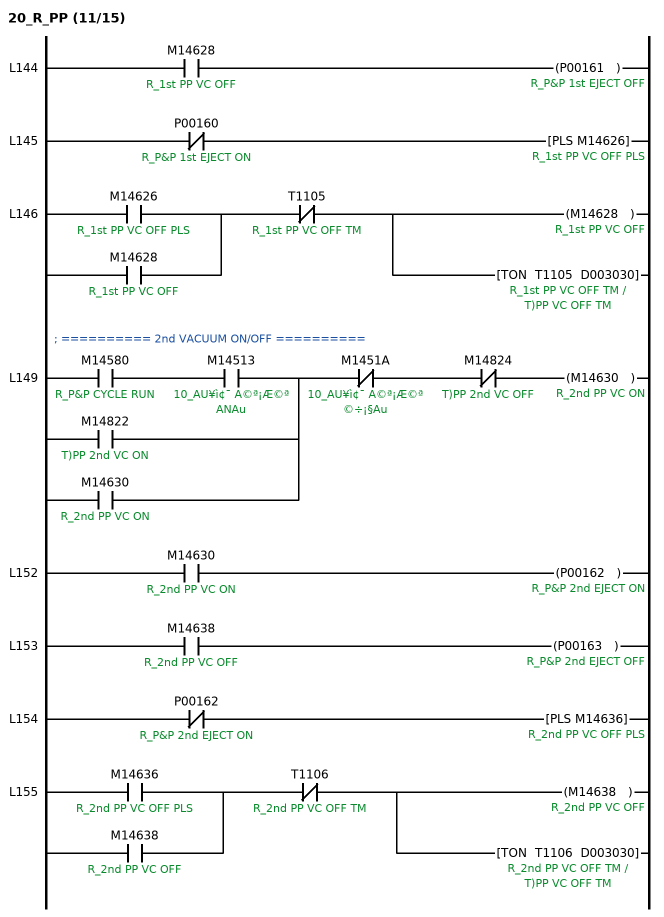
[picture p192: 20_R_PP rungs L144-L155]
; L144
LOAD      M14628	// R_1st PP VC OFF
OUT       P00161	// R_P&P 1st EJECT OFF
; L145
LOAD NOT  P00160	// R_P&P 1st EJECT ON
OUTP      M14626	// R_1st PP VC OFF PLS
; L146
LOAD      M14626	// R_1st PP VC OFF PLS
OR        M14628	// R_1st PP VC OFF
AND NOT   T1105	// R_1st PP VC OFF TM
OUT       M14628	// R_1st PP VC OFF
TON       T1105 D003030	// R_1st PP VC OFF TM / T)PP VC OFF TM
// ========== 2nd VACUUM ON/OFF ==========
; L149
LOAD      M14580	// R_P&P CYCLE RUN
AND       M14513	// 10_AU¥ì¢¯ A©ª¡Æ©ª ANAu
OR        M14822	// T)PP 2nd VC ON
OR        M14630	// R_2nd PP VC ON
AND NOT   M1451A	// 10_AU¥ì¢¯ A©ª¡Æ©ª ©÷¡§Au
AND NOT   M14824	// T)PP 2nd VC OFF
OUT       M14630	// R_2nd PP VC ON
; L152
LOAD      M14630	// R_2nd PP VC ON
OUT       P00162	// R_P&P 2nd EJECT ON
; L153
LOAD      M14638	// R_2nd PP VC OFF
OUT       P00163	// R_P&P 2nd EJECT OFF
; L154
LOAD NOT  P00162	// R_P&P 2nd EJECT ON
OUTP      M14636	// R_2nd PP VC OFF PLS
; L155
LOAD      M14636	// R_2nd PP VC OFF PLS
OR        M14638	// R_2nd PP VC OFF
AND NOT   T1106	// R_2nd PP VC OFF TM
OUT       M14638	// R_2nd PP VC OFF
TON       T1106 D003030	// R_2nd PP VC OFF TM / T)PP VC OFF TM

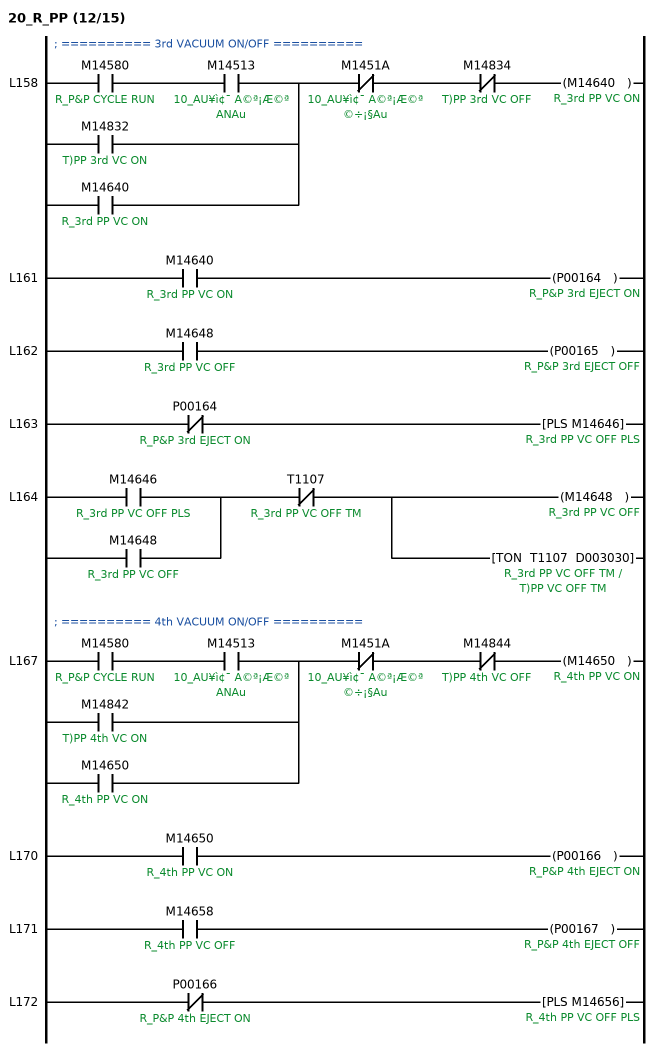
// ========== 3rd VACUUM ON/OFF ==========
; L158
LOAD      M14580	// R_P&P CYCLE RUN
AND       M14513	// 10_AU¥ì¢¯ A©ª¡Æ©ª ANAu
OR        M14832	// T)PP 3rd VC ON
OR        M14640	// R_3rd PP VC ON
AND NOT   M1451A	// 10_AU¥ì¢¯ A©ª¡Æ©ª ©÷¡§Au
AND NOT   M14834	// T)PP 3rd VC OFF
OUT       M14640	// R_3rd PP VC ON
; L161
LOAD      M14640	// R_3rd PP VC ON
OUT       P00164	// R_P&P 3rd EJECT ON
; L162
LOAD      M14648	// R_3rd PP VC OFF
OUT       P00165	// R_P&P 3rd EJECT OFF
; L163
LOAD NOT  P00164	// R_P&P 3rd EJECT ON
OUTP      M14646	// R_3rd PP VC OFF PLS
; L164
LOAD      M14646	// R_3rd PP VC OFF PLS
OR        M14648	// R_3rd PP VC OFF
AND NOT   T1107	// R_3rd PP VC OFF TM
OUT       M14648	// R_3rd PP VC OFF
TON       T1107 D003030	// R_3rd PP VC OFF TM / T)PP VC OFF TM
// ========== 4th VACUUM ON/OFF ==========
; L167
LOAD      M14580	// R_P&P CYCLE RUN
AND       M14513	// 10_AU¥ì¢¯ A©ª¡Æ©ª ANAu
OR        M14842	// T)PP 4th VC ON
OR        M14650	// R_4th PP VC ON
AND NOT   M1451A	// 10_AU¥ì¢¯ A©ª¡Æ©ª ©÷¡§Au
AND NOT   M14844	// T)PP 4th VC OFF
OUT       M14650	// R_4th PP VC ON
; L170
LOAD      M14650	// R_4th PP VC ON
OUT       P00166	// R_P&P 4th EJECT ON
; L171
LOAD      M14658	// R_4th PP VC OFF
OUT       P00167	// R_P&P 4th EJECT OFF
; L172
LOAD NOT  P00166	// R_P&P 4th EJECT ON
OUTP      M14656	// R_4th PP VC OFF PLS

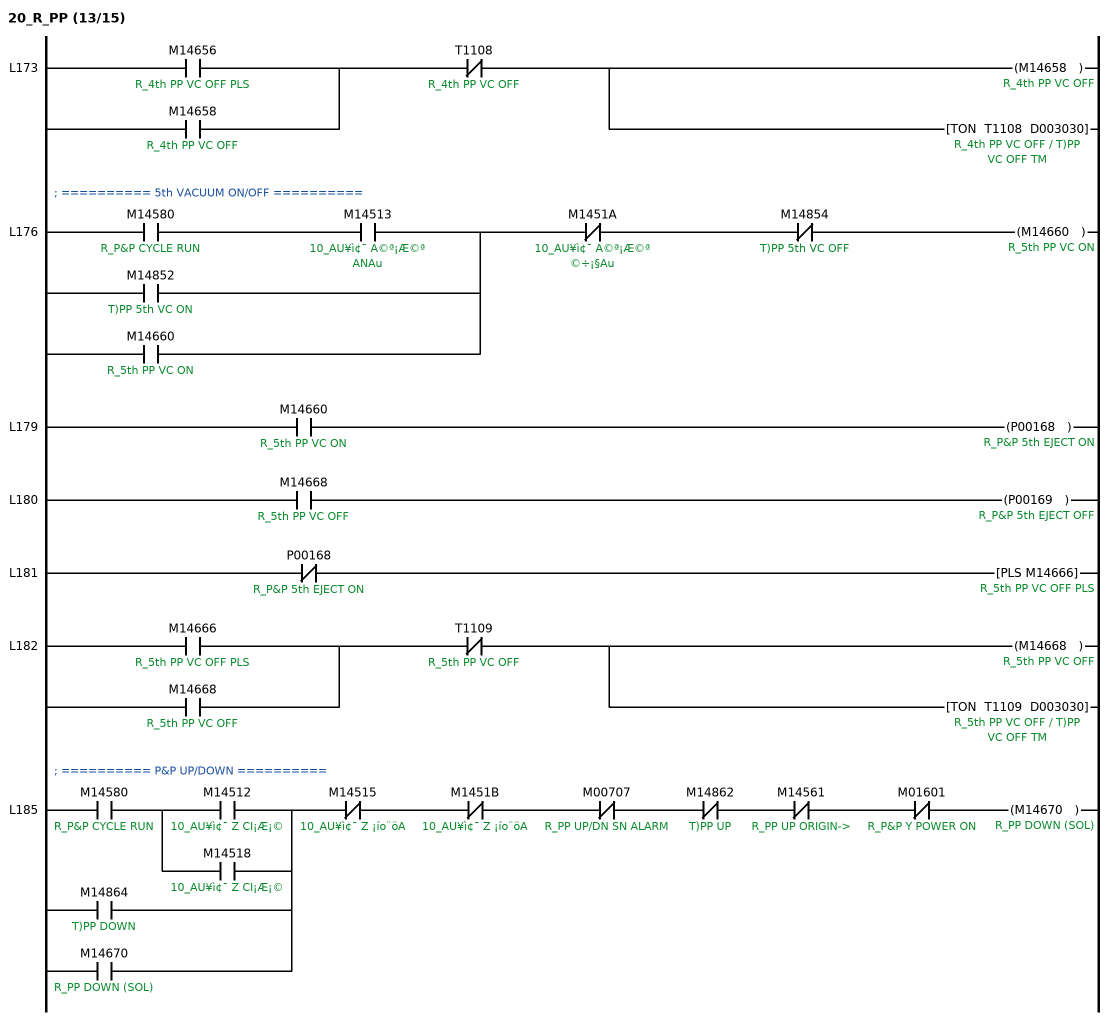
; L173
LOAD      M14656	// R_4th PP VC OFF PLS
OR        M14658	// R_4th PP VC OFF
AND NOT   T1108	// R_4th PP VC OFF
OUT       M14658	// R_4th PP VC OFF
TON       T1108 D003030	// R_4th PP VC OFF / T)PP VC OFF TM
// ========== 5th VACUUM ON/OFF ==========
; L176
LOAD      M14580	// R_P&P CYCLE RUN
AND       M14513	// 10_AU¥ì¢¯ A©ª¡Æ©ª ANAu
OR        M14852	// T)PP 5th VC ON
OR        M14660	// R_5th PP VC ON
AND NOT   M1451A	// 10_AU¥ì¢¯ A©ª¡Æ©ª ©÷¡§Au
AND NOT   M14854	// T)PP 5th VC OFF
OUT       M14660	// R_5th PP VC ON
; L179
LOAD      M14660	// R_5th PP VC ON
OUT       P00168	// R_P&P 5th EJECT ON
; L180
LOAD      M14668	// R_5th PP VC OFF
OUT       P00169	// R_P&P 5th EJECT OFF
; L181
LOAD NOT  P00168	// R_P&P 5th EJECT ON
OUTP      M14666	// R_5th PP VC OFF PLS
; L182
LOAD      M14666	// R_5th PP VC OFF PLS
OR        M14668	// R_5th PP VC OFF
AND NOT   T1109	// R_5th PP VC OFF
OUT       M14668	// R_5th PP VC OFF
TON       T1109 D003030	// R_5th PP VC OFF / T)PP VC OFF TM
// ========== P&P UP/DOWN ==========
; L185
LOAD      M14580	// R_P&P CYCLE RUN
LOAD      M14512	// 10_AU¥ì¢¯ Z CI¡Æ¡©
OR        M14518	// 10_AU¥ì¢¯ Z CI¡Æ¡©
AND LOAD
OR        M14864	// T)PP DOWN
OR        M14670	// R_PP DOWN (SOL)
AND NOT   M14515	// 10_AU¥ì¢¯ Z ¡ío¨öA
AND NOT   M1451B	// 10_AU¥ì¢¯ Z ¡ío¨öA
AND NOT   M00707	// R_PP UP/DN SN ALARM
AND NOT   M14862	// T)PP UP
AND NOT   M14561	// R_PP UP ORIGIN->
AND NOT   M01601	// R_P&P Y POWER ON
OUT       M14670	// R_PP DOWN (SOL)

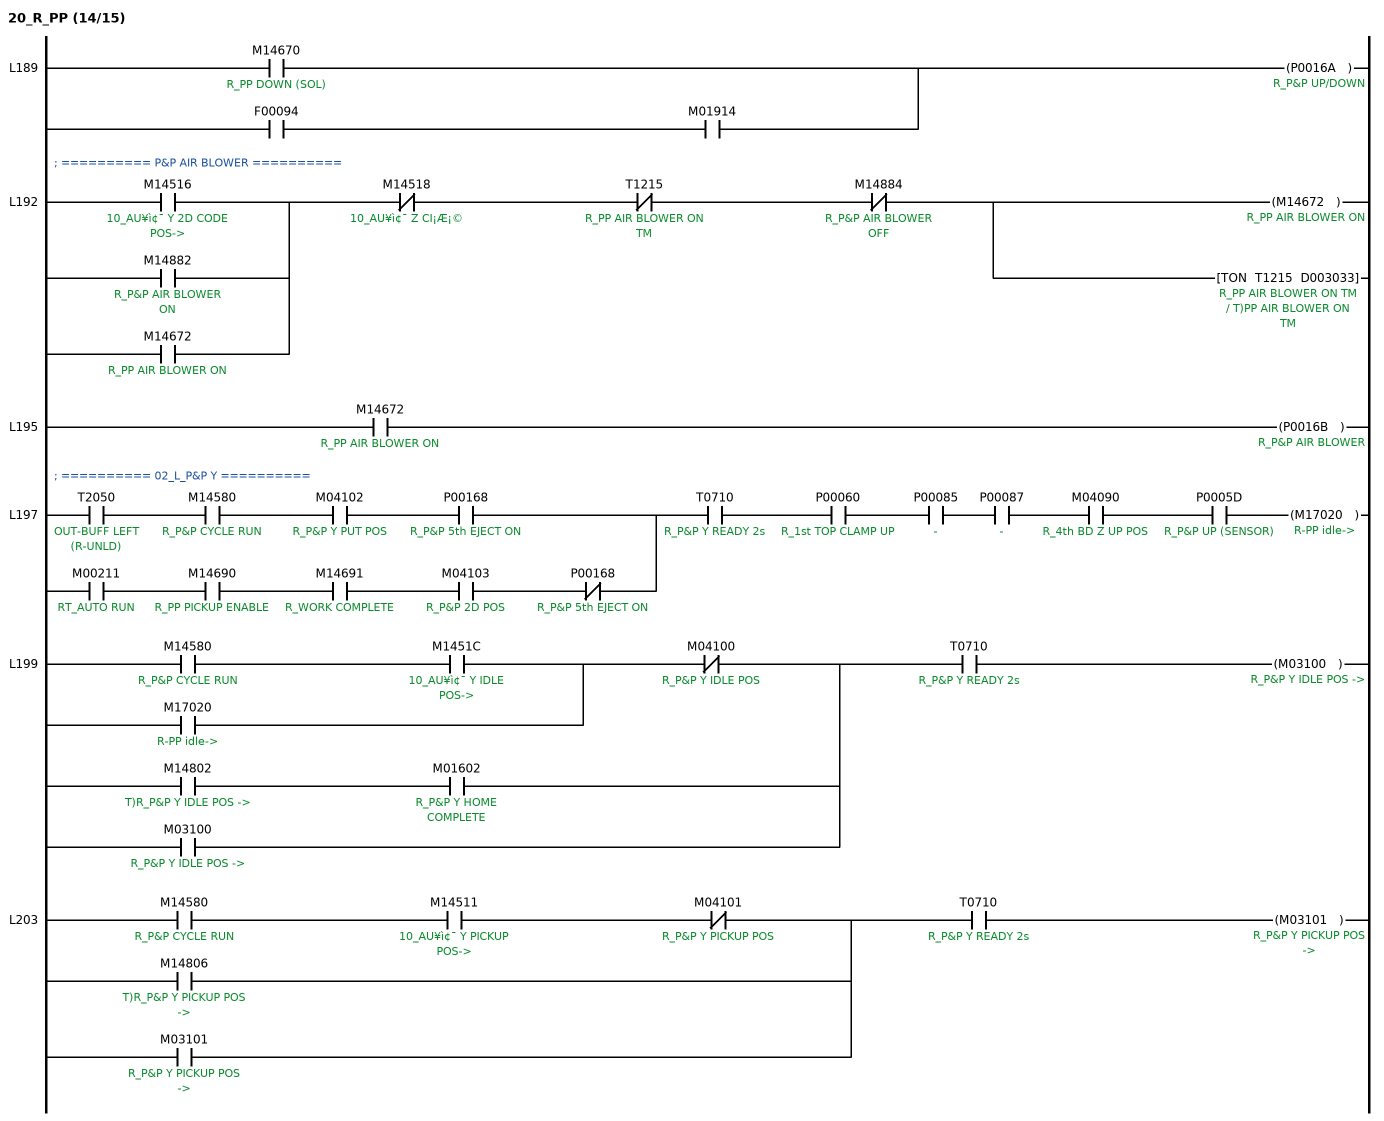
; L189
LOAD      M14670	// R_PP DOWN (SOL)
LOAD      F00094
AND       M01914
OR LOAD
OUT       P0016A	// R_P&P UP/DOWN
// ========== P&P AIR BLOWER ==========
; L192
LOAD      M14516	// 10_AU¥ì¢¯ Y 2D CODE POS->
OR        M14882	// R_P&P AIR BLOWER ON
OR        M14672	// R_PP AIR BLOWER ON
AND NOT   M14518	// 10_AU¥ì¢¯ Z CI¡Æ¡©
AND NOT   T1215	// R_PP AIR BLOWER ON TM
AND NOT   M14884	// R_P&P AIR BLOWER OFF
OUT       M14672	// R_PP AIR BLOWER ON
TON       T1215 D003033	// R_PP AIR BLOWER ON TM / T)PP AIR BLOWER ON TM
; L195
LOAD      M14672	// R_PP AIR BLOWER ON
OUT       P0016B	// R_P&P AIR BLOWER
// ========== 02_L_P&P Y ==========
; L197
LOAD      T2050	// OUT-BUFF LEFT (R-UNLD)
AND       M14580	// R_P&P CYCLE RUN
AND       M04102	// R_P&P Y PUT POS
AND       P00168	// R_P&P 5th EJECT ON
LOAD      M00211	// RT_AUTO RUN
AND       M14690	// R_PP PICKUP ENABLE
AND       M14691	// R_WORK COMPLETE
AND       M04103	// R_P&P 2D POS
AND NOT   P00168	// R_P&P 5th EJECT ON
OR LOAD
AND       T0710	// R_P&P Y READY 2s
AND       P00060	// R_1st TOP CLAMP UP
AND       P00085	// -
AND       P00087	// -
AND       M04090	// R_4th BD Z UP POS
AND       P0005D	// R_P&P UP (SENSOR)
OUT       M17020	// R-PP idle->
; L199
LOAD      M14580	// R_P&P CYCLE RUN
AND       M1451C	// 10_AU¥ì¢¯ Y IDLE POS->
OR        M17020	// R-PP idle->
AND NOT   M04100	// R_P&P Y IDLE POS
LOAD      M14802	// T)R_P&P Y IDLE POS ->
AND       M01602	// R_P&P Y HOME COMPLETE
OR LOAD
OR        M03100	// R_P&P Y IDLE POS ->
AND       T0710	// R_P&P Y READY 2s
OUT       M03100	// R_P&P Y IDLE POS ->
; L203
LOAD      M14580	// R_P&P CYCLE RUN
AND       M14511	// 10_AU¥ì¢¯ Y PICKUP POS->
AND NOT   M04101	// R_P&P Y PICKUP POS
OR        M14806	// T)R_P&P Y PICKUP POS ->
OR        M03101	// R_P&P Y PICKUP POS ->
AND       T0710	// R_P&P Y READY 2s
OUT       M03101	// R_P&P Y PICKUP POS ->

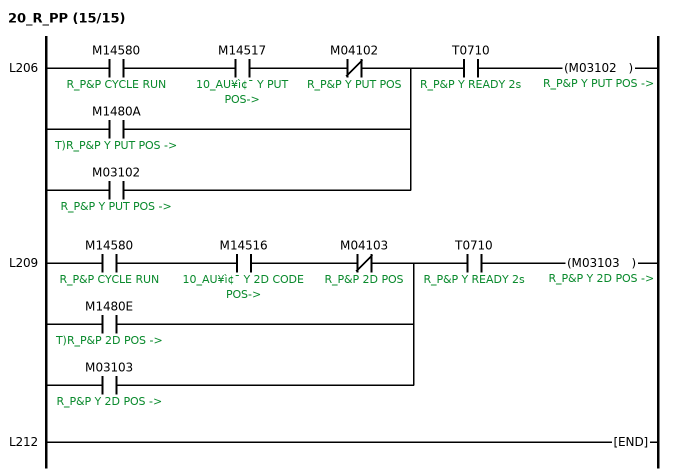
; L206
LOAD      M14580	// R_P&P CYCLE RUN
AND       M14517	// 10_AU¥ì¢¯ Y PUT POS->
AND NOT   M04102	// R_P&P Y PUT POS
OR        M1480A	// T)R_P&P Y PUT POS ->
OR        M03102	// R_P&P Y PUT POS ->
AND       T0710	// R_P&P Y READY 2s
OUT       M03102	// R_P&P Y PUT POS ->
; L209
LOAD      M14580	// R_P&P CYCLE RUN
AND       M14516	// 10_AU¥ì¢¯ Y 2D CODE POS->
AND NOT   M04103	// R_P&P 2D POS
OR        M1480E	// T)R_P&P 2D POS ->
OR        M03103	// R_P&P Y 2D POS ->
AND       T0710	// R_P&P Y READY 2s
OUT       M03103	// R_P&P Y 2D POS ->
; L212
END

PROGRAM 30_IN_LR_BUFFER (task: ¨ö¨¬A¥ì CA¡¤I¡¾¡¿¡¤¡Í)

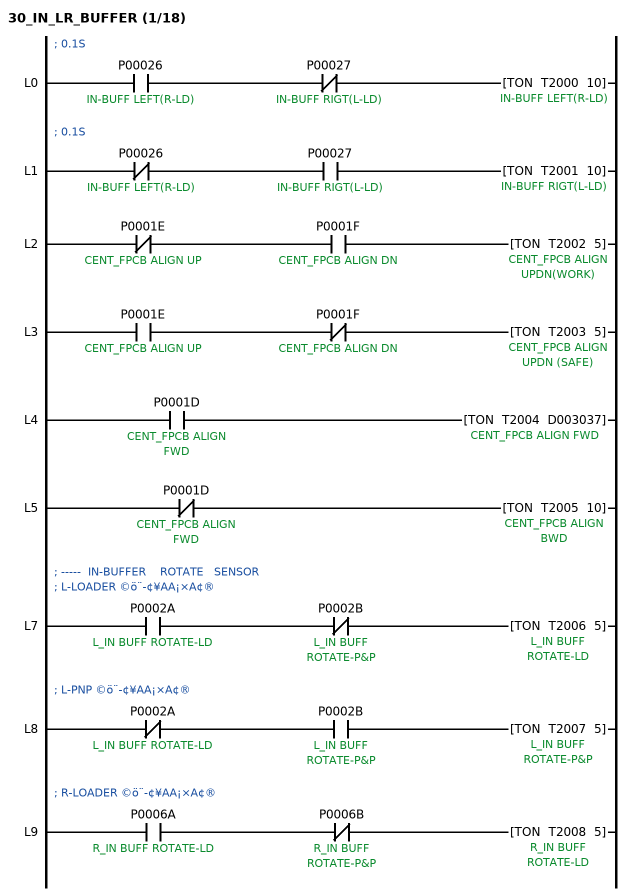
; L0
LOAD      P00026	// IN-BUFF LEFT(R-LD)
AND NOT   P00027	// IN-BUFF RIGT(L-LD)
TON       T2000 10	// IN-BUFF LEFT(R-LD)
// output comment: 0.1S
; L1
LOAD NOT  P00026	// IN-BUFF LEFT(R-LD)
AND       P00027	// IN-BUFF RIGT(L-LD)
TON       T2001 10	// IN-BUFF RIGT(L-LD)
// output comment: 0.1S
; L2
LOAD NOT  P0001E	// CENT_FPCB ALIGN UP
AND       P0001F	// CENT_FPCB ALIGN DN
TON       T2002 5	// CENT_FPCB ALIGN UPDN(WORK)
; L3
LOAD      P0001E	// CENT_FPCB ALIGN UP
AND NOT   P0001F	// CENT_FPCB ALIGN DN
TON       T2003 5	// CENT_FPCB ALIGN UPDN (SAFE)
; L4
LOAD      P0001D	// CENT_FPCB ALIGN FWD
TON       T2004 D003037	// CENT_FPCB ALIGN FWD
; L5
LOAD NOT  P0001D	// CENT_FPCB ALIGN FWD
TON       T2005 10	// CENT_FPCB ALIGN BWD
// -----  IN-BUFFER    ROTATE   SENSOR
; L7
LOAD      P0002A	// L_IN BUFF ROTATE-LD
AND NOT   P0002B	// L_IN BUFF ROTATE-P&P
TON       T2006 5	// L_IN BUFF ROTATE-LD
// output comment: L-LOADER ©ö¨­¢¥AA¡×A¢®
; L8
LOAD NOT  P0002A	// L_IN BUFF ROTATE-LD
AND       P0002B	// L_IN BUFF ROTATE-P&P
TON       T2007 5	// L_IN BUFF ROTATE-P&P
// output comment: L-PNP ©ö¨­¢¥AA¡×A¢®
; L9
LOAD      P0006A	// R_IN BUFF ROTATE-LD
AND NOT   P0006B	// R_IN BUFF ROTATE-P&P
TON       T2008 5	// R_IN BUFF ROTATE-LD
// output comment: R-LOADER ©ö¨­¢¥AA¡×A¢®

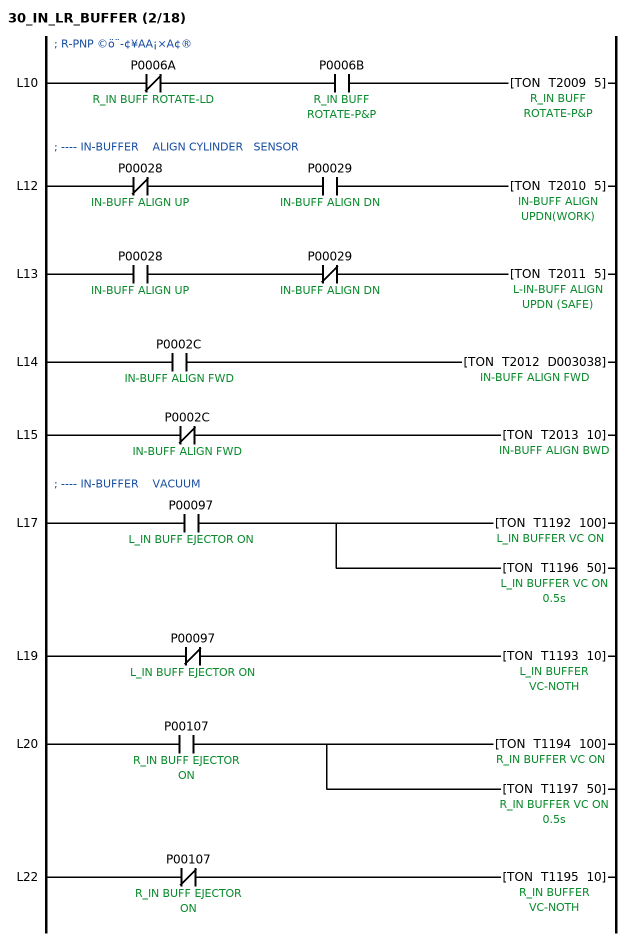
; L10
LOAD NOT  P0006A	// R_IN BUFF ROTATE-LD
AND       P0006B	// R_IN BUFF ROTATE-P&P
TON       T2009 5	// R_IN BUFF ROTATE-P&P
// output comment: R-PNP ©ö¨­¢¥AA¡×A¢®
// ---- IN-BUFFER    ALIGN CYLINDER   SENSOR
; L12
LOAD NOT  P00028	// IN-BUFF ALIGN UP
AND       P00029	// IN-BUFF ALIGN DN
TON       T2010 5	// IN-BUFF ALIGN UPDN(WORK)
; L13
LOAD      P00028	// IN-BUFF ALIGN UP
AND NOT   P00029	// IN-BUFF ALIGN DN
TON       T2011 5	// L-IN-BUFF ALIGN UPDN (SAFE)
; L14
LOAD      P0002C	// IN-BUFF ALIGN FWD
TON       T2012 D003038	// IN-BUFF ALIGN FWD
; L15
LOAD NOT  P0002C	// IN-BUFF ALIGN FWD
TON       T2013 10	// IN-BUFF ALIGN BWD
// ---- IN-BUFFER    VACUUM
; L17
LOAD      P00097	// L_IN BUFF EJECTOR ON
TON       T1192 100	// L_IN BUFFER VC ON
TON       T1196 50	// L_IN BUFFER VC ON 0.5s
; L19
LOAD NOT  P00097	// L_IN BUFF EJECTOR ON
TON       T1193 10	// L_IN BUFFER VC-NOTH
; L20
LOAD      P00107	// R_IN BUFF EJECTOR ON
TON       T1194 100	// R_IN BUFFER VC ON
TON       T1197 50	// R_IN BUFFER VC ON 0.5s
; L22
LOAD NOT  P00107	// R_IN BUFF EJECTOR ON
TON       T1195 10	// R_IN BUFFER VC-NOTH

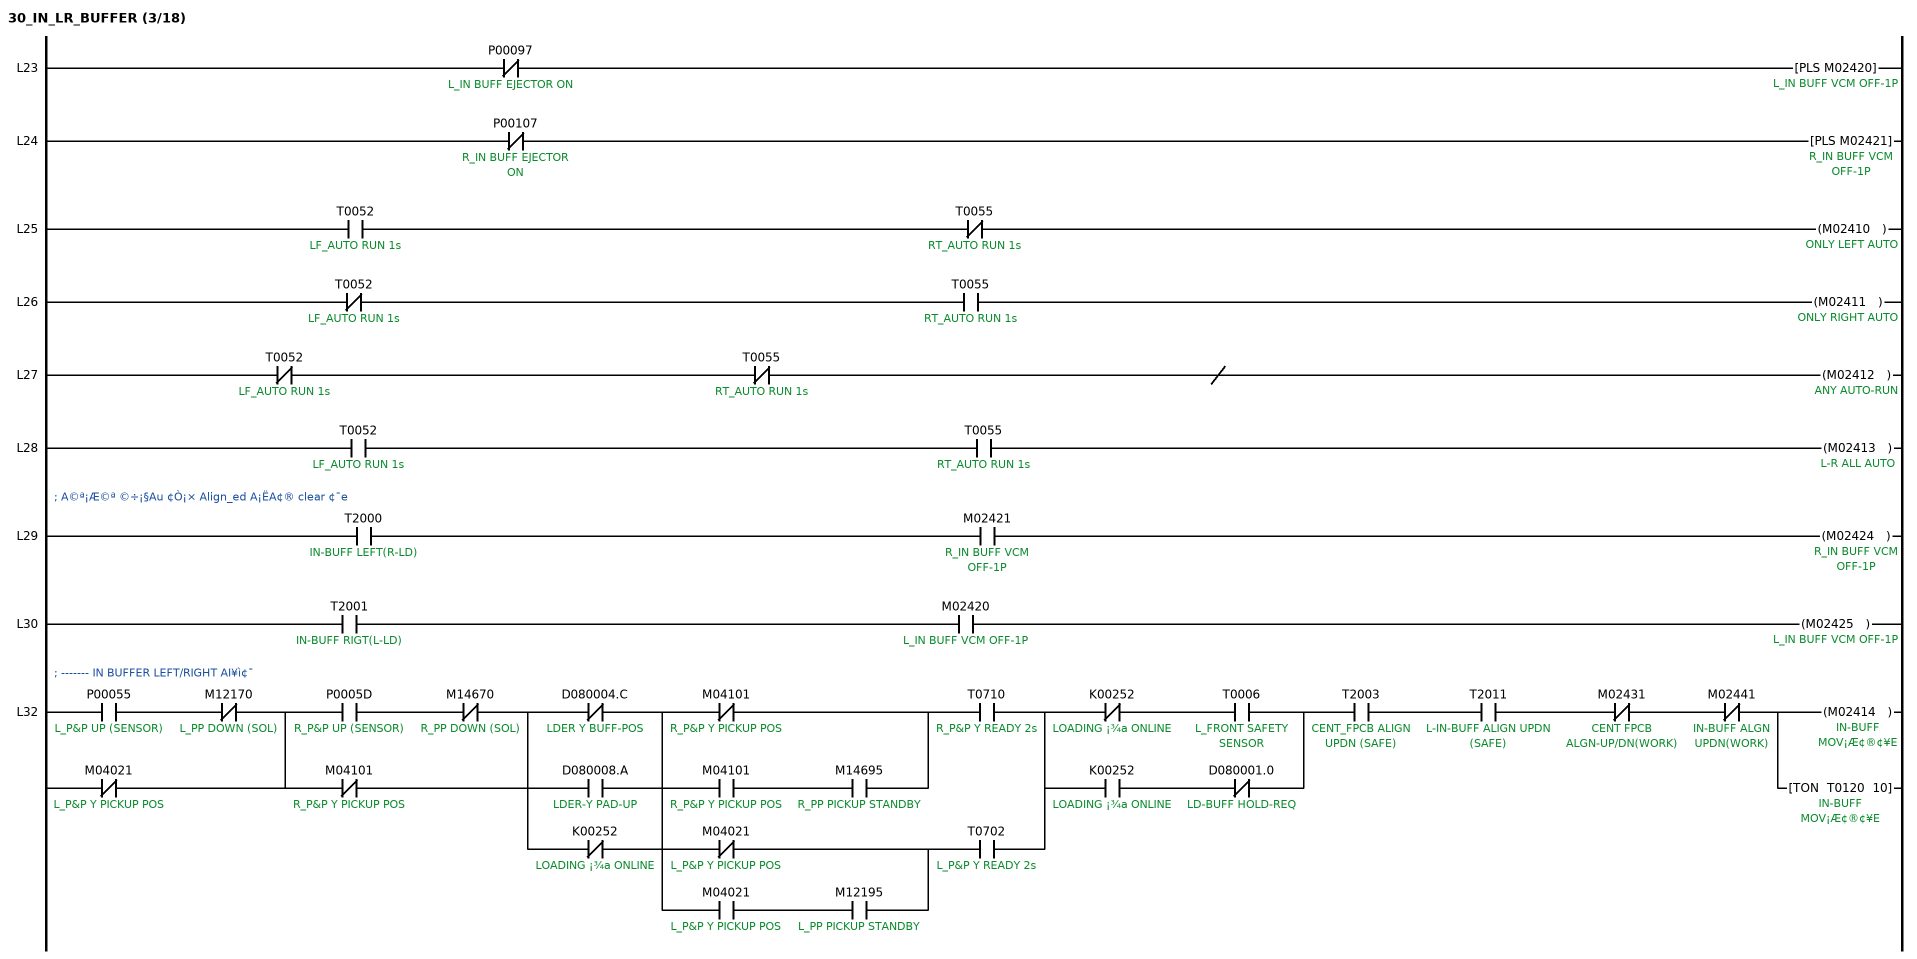
; L23
LOAD NOT  P00097	// L_IN BUFF EJECTOR ON
OUTP      M02420	// L_IN BUFF VCM OFF-1P
; L24
LOAD NOT  P00107	// R_IN BUFF EJECTOR ON
OUTP      M02421	// R_IN BUFF VCM OFF-1P
; L25
LOAD      T0052	// LF_AUTO RUN 1s
AND NOT   T0055	// RT_AUTO RUN 1s
OUT       M02410	// ONLY LEFT AUTO
; L26
LOAD NOT  T0052	// LF_AUTO RUN 1s
AND       T0055	// RT_AUTO RUN 1s
OUT       M02411	// ONLY RIGHT AUTO
; L27
LOAD NOT  T0052	// LF_AUTO RUN 1s
AND NOT   T0055	// RT_AUTO RUN 1s
NOT
OUT       M02412	// ANY AUTO-RUN
; L28
LOAD      T0052	// LF_AUTO RUN 1s
AND       T0055	// RT_AUTO RUN 1s
OUT       M02413	// L-R ALL AUTO
; L29
LOAD      T2000	// IN-BUFF LEFT(R-LD)
AND       M02421	// R_IN BUFF VCM OFF-1P
OUT       M02424	// R_IN BUFF VCM OFF-1P
// output comment: A©ª¡Æ©ª ©÷¡§Au ¢Ò¡× Align_ed A¡ËA¢® clear ¢¯e
; L30
LOAD      T2001	// IN-BUFF RIGT(L-LD)
AND       M02420	// L_IN BUFF VCM OFF-1P
OUT       M02425	// L_IN BUFF VCM OFF-1P
// ------- IN BUFFER LEFT/RIGHT AI¥ì¢¯
; L32
LOAD      P00055	// L_P&P UP (SENSOR)
AND NOT   M12170	// L_PP DOWN (SOL)
OR NOT    M04021	// L_P&P Y PICKUP POS
LOAD      P0005D	// R_P&P UP (SENSOR)
AND NOT   M14670	// R_PP DOWN (SOL)
OR NOT    M04101	// R_P&P Y PICKUP POS
AND LOAD
LOAD NOT  D080004.C	// LDER Y BUFF-POS
OR        D080008.A	// LDER-Y PAD-UP
OR NOT    K00252	// LOADING ¡¾a ONLINE
AND LOAD
LOAD NOT  M04101	// R_P&P Y PICKUP POS
LOAD      M04101	// R_P&P Y PICKUP POS
AND       M14695	// R_PP PICKUP STANDBY
OR LOAD
AND       T0710	// R_P&P Y READY 2s
LOAD NOT  M04021	// L_P&P Y PICKUP POS
LOAD      M04021	// L_P&P Y PICKUP POS
AND       M12195	// L_PP PICKUP STANDBY
OR LOAD
AND       T0702	// L_P&P Y READY 2s
OR LOAD
AND LOAD
LOAD NOT  K00252	// LOADING ¡¾a ONLINE
AND       T0006	// L_FRONT SAFETY SENSOR
LOAD      K00252	// LOADING ¡¾a ONLINE
AND NOT   D080001.0	// LD-BUFF HOLD-REQ
OR LOAD
AND LOAD
AND       T2003	// CENT_FPCB ALIGN UPDN (SAFE)
AND       T2011	// L-IN-BUFF ALIGN UPDN (SAFE)
AND NOT   M02431	// CENT FPCB ALGN-UP/DN(WORK)
AND NOT   M02441	// IN-BUFF ALGN UPDN(WORK)
OUT       M02414	// IN-BUFF MOV¡Æ¢®¢¥E
TON       T0120 10	// IN-BUFF MOV¡Æ¢®¢¥E

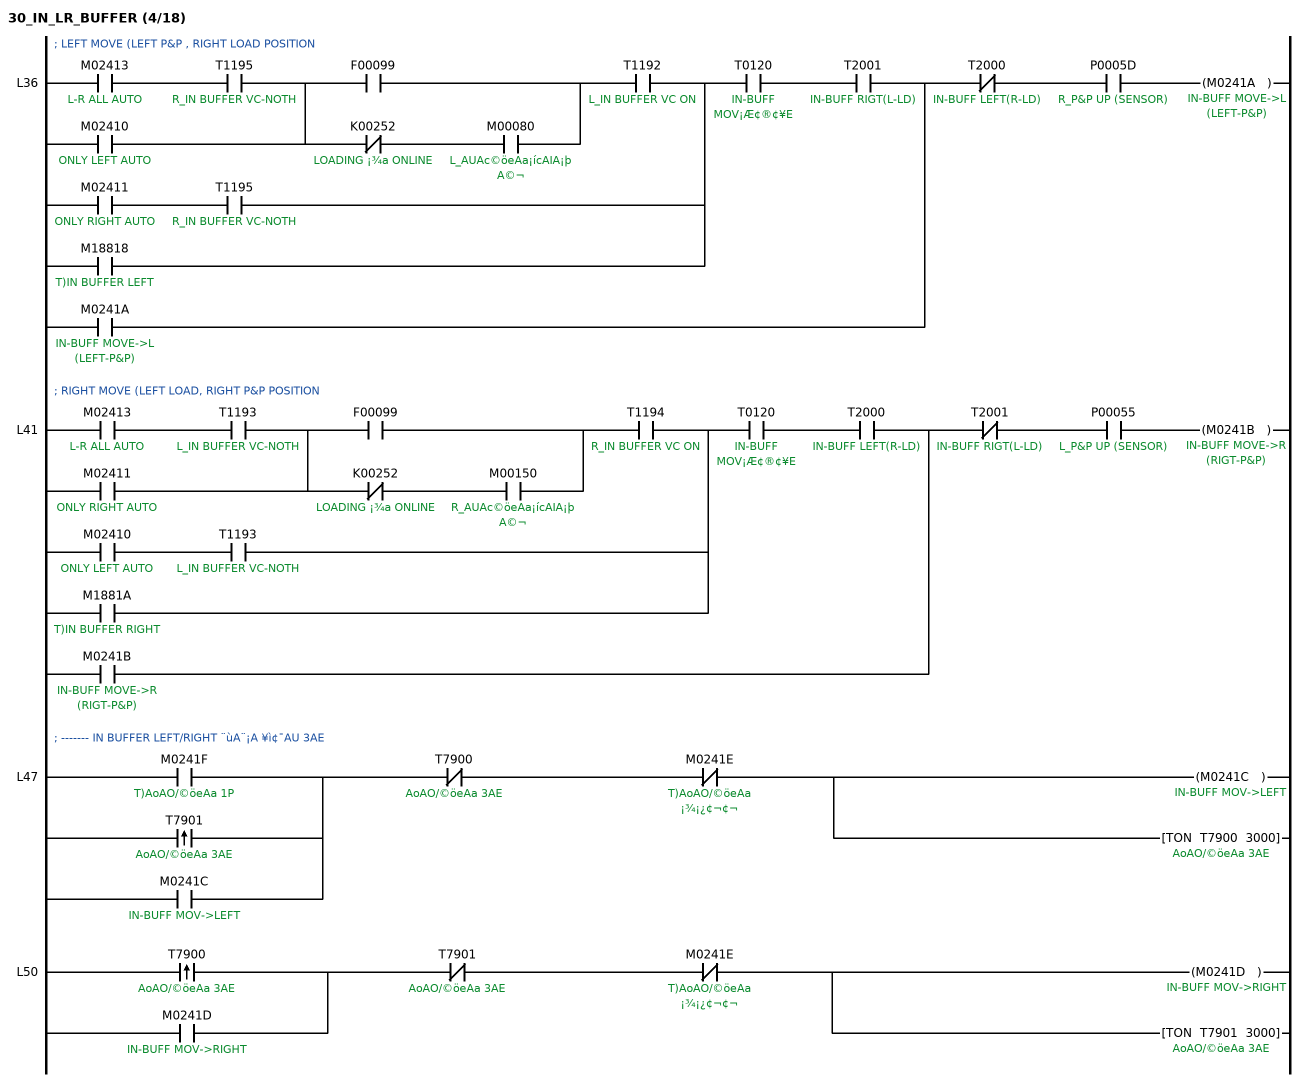
; L36
LOAD      M02413	// L-R ALL AUTO
AND       T1195	// R_IN BUFFER VC-NOTH
OR        M02410	// ONLY LEFT AUTO
LOAD      F00099
LOAD NOT  K00252	// LOADING ¡¾a ONLINE
AND       M00080	// L_AUAc©öeAa¡ícAIA¡þA©¬
OR LOAD
AND LOAD
AND       T1192	// L_IN BUFFER VC ON
LOAD      M02411	// ONLY RIGHT AUTO
AND       T1195	// R_IN BUFFER VC-NOTH
OR LOAD
OR        M18818	// T)IN BUFFER LEFT
AND       T0120	// IN-BUFF MOV¡Æ¢®¢¥E
AND       T2001	// IN-BUFF RIGT(L-LD)
OR        M0241A	// IN-BUFF MOVE->L (LEFT-P&P)
AND NOT   T2000	// IN-BUFF LEFT(R-LD)
AND       P0005D	// R_P&P UP (SENSOR)
OUT       M0241A	// IN-BUFF MOVE->L (LEFT-P&P)
// output comment: LEFT MOVE (LEFT P&P , RIGHT LOAD POSITION
; L41
LOAD      M02413	// L-R ALL AUTO
AND       T1193	// L_IN BUFFER VC-NOTH
OR        M02411	// ONLY RIGHT AUTO
LOAD      F00099
LOAD NOT  K00252	// LOADING ¡¾a ONLINE
AND       M00150	// R_AUAc©öeAa¡ícAIA¡þA©¬
OR LOAD
AND LOAD
AND       T1194	// R_IN BUFFER VC ON
LOAD      M02410	// ONLY LEFT AUTO
AND       T1193	// L_IN BUFFER VC-NOTH
OR LOAD
OR        M1881A	// T)IN BUFFER RIGHT
AND       T0120	// IN-BUFF MOV¡Æ¢®¢¥E
AND       T2000	// IN-BUFF LEFT(R-LD)
OR        M0241B	// IN-BUFF MOVE->R (RIGT-P&P)
AND NOT   T2001	// IN-BUFF RIGT(L-LD)
AND       P00055	// L_P&P UP (SENSOR)
OUT       M0241B	// IN-BUFF MOVE->R (RIGT-P&P)
// output comment: RIGHT MOVE (LEFT LOAD, RIGHT P&P POSITION
// ------- IN BUFFER LEFT/RIGHT ¨ùA¨¡A ¥ì¢¯AU 3AE
; L47
LOAD      M0241F	// T)AoAO/©öeAa 1P
ORP       T7901	// AoAO/©öeAa 3AE
OR        M0241C	// IN-BUFF MOV->LEFT
AND NOT   T7900	// AoAO/©öeAa 3AE
AND NOT   M0241E	// T)AoAO/©öeAa ¡¾¡¿¢¬¢¬
OUT       M0241C	// IN-BUFF MOV->LEFT
TON       T7900 3000	// AoAO/©öeAa 3AE
; L50
LOADP     T7900	// AoAO/©öeAa 3AE
OR        M0241D	// IN-BUFF MOV->RIGHT
AND NOT   T7901	// AoAO/©öeAa 3AE
AND NOT   M0241E	// T)AoAO/©öeAa ¡¾¡¿¢¬¢¬
OUT       M0241D	// IN-BUFF MOV->RIGHT
TON       T7901 3000	// AoAO/©öeAa 3AE

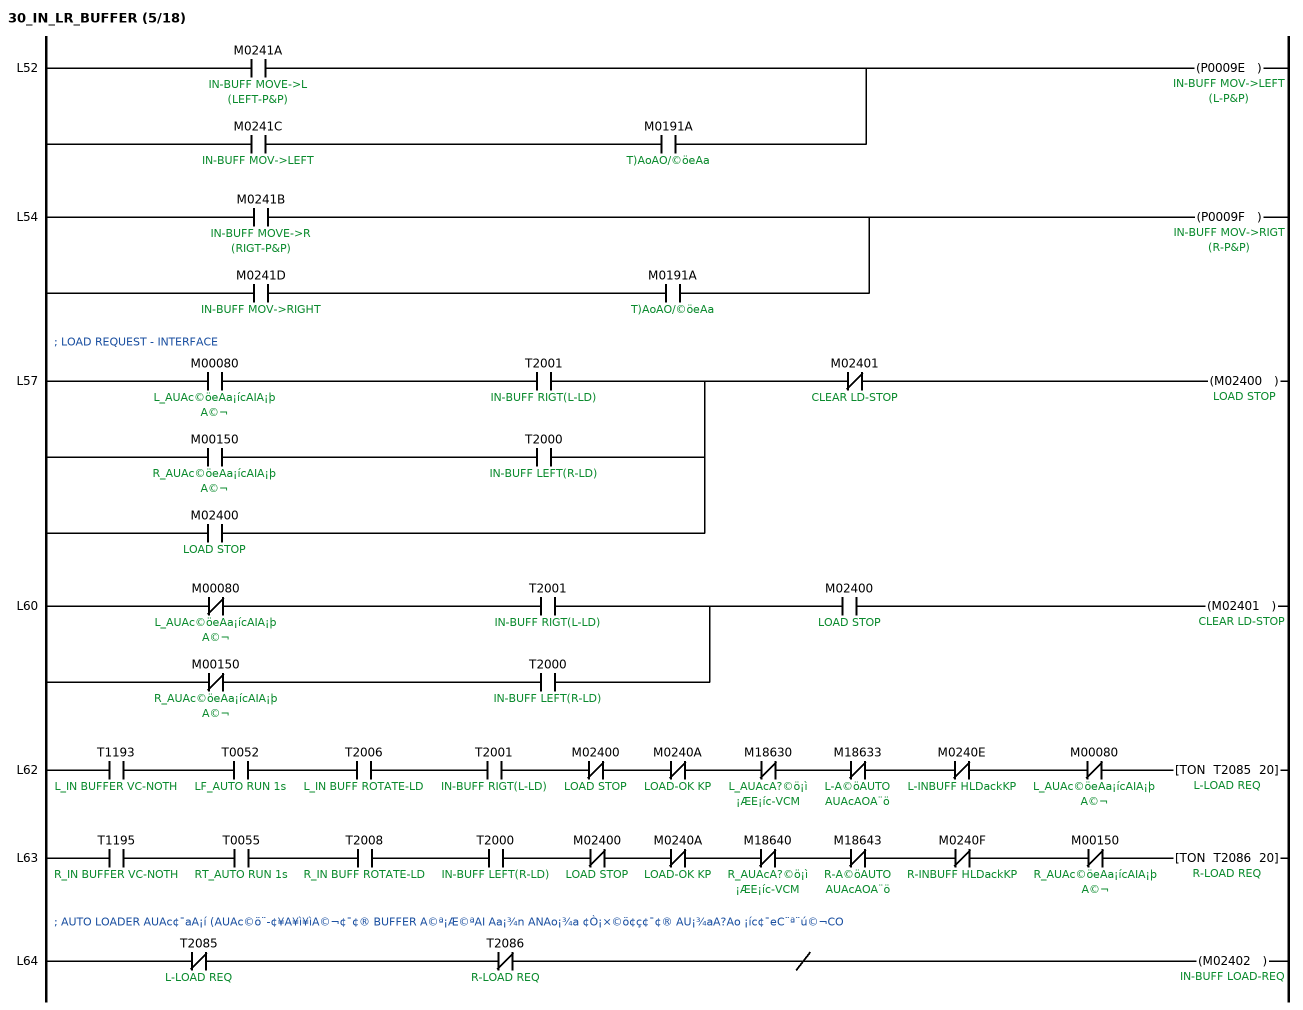
; L52
LOAD      M0241A	// IN-BUFF MOVE->L (LEFT-P&P)
LOAD      M0241C	// IN-BUFF MOV->LEFT
AND       M0191A	// T)AoAO/©öeAa
OR LOAD
OUT       P0009E	// IN-BUFF MOV->LEFT (L-P&P)
; L54
LOAD      M0241B	// IN-BUFF MOVE->R (RIGT-P&P)
LOAD      M0241D	// IN-BUFF MOV->RIGHT
AND       M0191A	// T)AoAO/©öeAa
OR LOAD
OUT       P0009F	// IN-BUFF MOV->RIGT (R-P&P)
// LOAD REQUEST - INTERFACE
; L57
LOAD      M00080	// L_AUAc©öeAa¡ícAIA¡þA©¬
AND       T2001	// IN-BUFF RIGT(L-LD)
LOAD      M00150	// R_AUAc©öeAa¡ícAIA¡þA©¬
AND       T2000	// IN-BUFF LEFT(R-LD)
OR LOAD
OR        M02400	// LOAD STOP
AND NOT   M02401	// CLEAR LD-STOP
OUT       M02400	// LOAD STOP
; L60
LOAD NOT  M00080	// L_AUAc©öeAa¡ícAIA¡þA©¬
AND       T2001	// IN-BUFF RIGT(L-LD)
LOAD NOT  M00150	// R_AUAc©öeAa¡ícAIA¡þA©¬
AND       T2000	// IN-BUFF LEFT(R-LD)
OR LOAD
AND       M02400	// LOAD STOP
OUT       M02401	// CLEAR LD-STOP
; L62
LOAD      T1193	// L_IN BUFFER VC-NOTH
AND       T0052	// LF_AUTO RUN 1s
AND       T2006	// L_IN BUFF ROTATE-LD
AND       T2001	// IN-BUFF RIGT(L-LD)
AND NOT   M02400	// LOAD STOP
AND NOT   M0240A	// LOAD-OK KP
AND NOT   M18630	// L_AUAcA?©ö¡ì ¡ÆE¡íc-VCM
AND NOT   M18633	// L-A©öAUTO AUAcAOA¨ö
AND NOT   M0240E	// L-INBUFF HLDackKP
AND NOT   M00080	// L_AUAc©öeAa¡ícAIA¡þA©¬
TON       T2085 20	// L-LOAD REQ
; L63
LOAD      T1195	// R_IN BUFFER VC-NOTH
AND       T0055	// RT_AUTO RUN 1s
AND       T2008	// R_IN BUFF ROTATE-LD
AND       T2000	// IN-BUFF LEFT(R-LD)
AND NOT   M02400	// LOAD STOP
AND NOT   M0240A	// LOAD-OK KP
AND NOT   M18640	// R_AUAcA?©ö¡ì ¡ÆE¡íc-VCM
AND NOT   M18643	// R-A©öAUTO AUAcAOA¨ö
AND NOT   M0240F	// R-INBUFF HLDackKP
AND NOT   M00150	// R_AUAc©öeAa¡ícAIA¡þA©¬
TON       T2086 20	// R-LOAD REQ
; L64
LOAD NOT  T2085	// L-LOAD REQ
AND NOT   T2086	// R-LOAD REQ
NOT
OUT       M02402	// IN-BUFF LOAD-REQ
// output comment: AUTO LOADER AUAc¢¯aA¡í (AUAc©ö¨­¢¥A¥ì¥ìA©¬¢¯¢® BUFFER A©ª¡Æ©ªAI Aa¡¾n ANAo¡¾a ¢Ò¡×©ö¢ç¢¯¢® AU¡¾aA?Ao ¡íc¢¯eC¨ª¨ú©¬CO

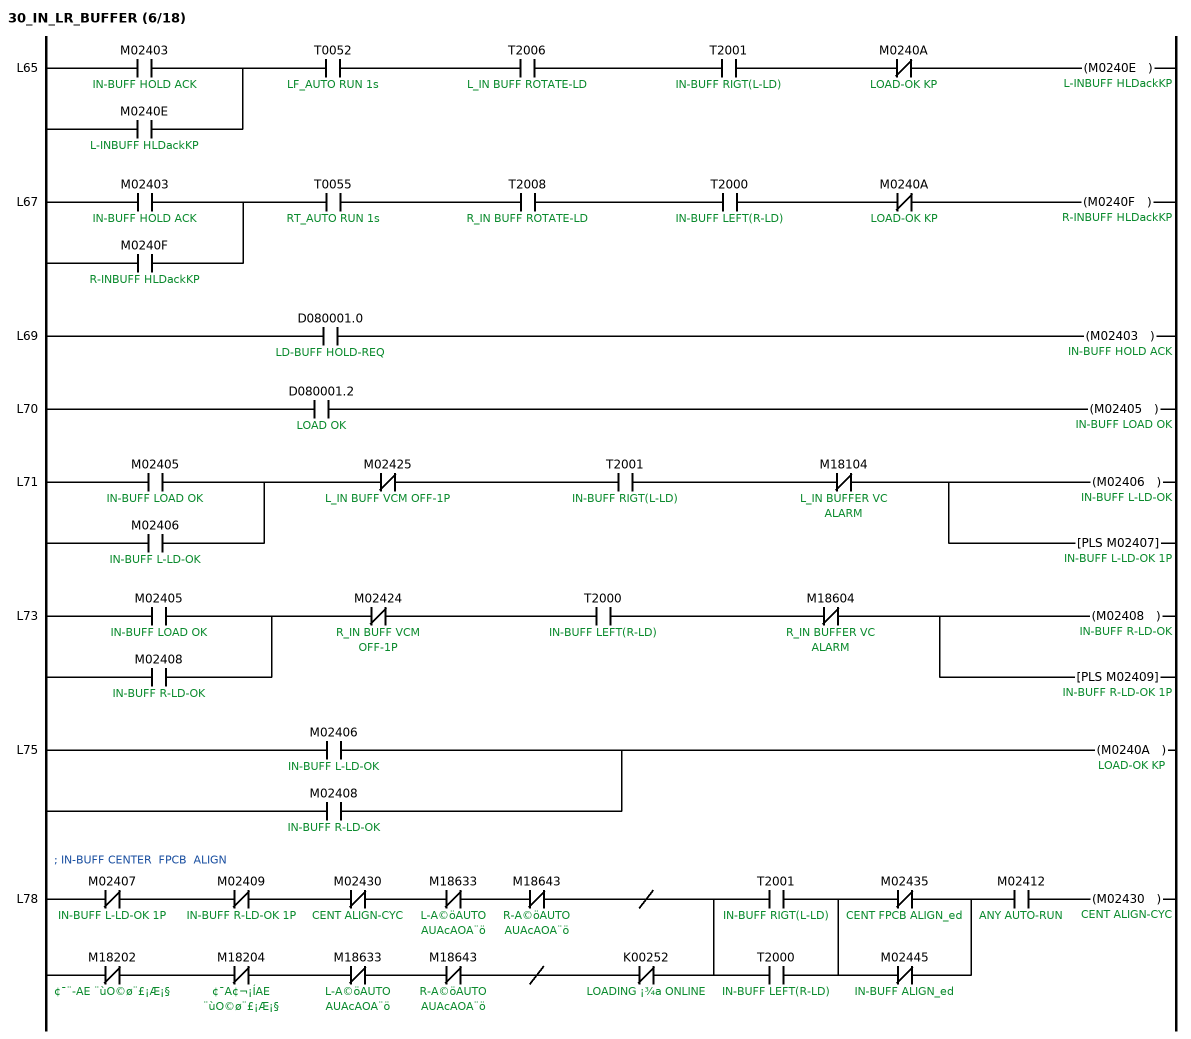
; L65
LOAD      M02403	// IN-BUFF HOLD ACK
OR        M0240E	// L-INBUFF HLDackKP
AND       T0052	// LF_AUTO RUN 1s
AND       T2006	// L_IN BUFF ROTATE-LD
AND       T2001	// IN-BUFF RIGT(L-LD)
AND NOT   M0240A	// LOAD-OK KP
OUT       M0240E	// L-INBUFF HLDackKP
; L67
LOAD      M02403	// IN-BUFF HOLD ACK
OR        M0240F	// R-INBUFF HLDackKP
AND       T0055	// RT_AUTO RUN 1s
AND       T2008	// R_IN BUFF ROTATE-LD
AND       T2000	// IN-BUFF LEFT(R-LD)
AND NOT   M0240A	// LOAD-OK KP
OUT       M0240F	// R-INBUFF HLDackKP
; L69
LOAD      D080001.0	// LD-BUFF HOLD-REQ
OUT       M02403	// IN-BUFF HOLD ACK
; L70
LOAD      D080001.2	// LOAD OK
OUT       M02405	// IN-BUFF LOAD OK
; L71
LOAD      M02405	// IN-BUFF LOAD OK
OR        M02406	// IN-BUFF L-LD-OK
AND NOT   M02425	// L_IN BUFF VCM OFF-1P
AND       T2001	// IN-BUFF RIGT(L-LD)
AND NOT   M18104	// L_IN BUFFER VC ALARM
OUT       M02406	// IN-BUFF L-LD-OK
OUTP      M02407	// IN-BUFF L-LD-OK 1P
; L73
LOAD      M02405	// IN-BUFF LOAD OK
OR        M02408	// IN-BUFF R-LD-OK
AND NOT   M02424	// R_IN BUFF VCM OFF-1P
AND       T2000	// IN-BUFF LEFT(R-LD)
AND NOT   M18604	// R_IN BUFFER VC ALARM
OUT       M02408	// IN-BUFF R-LD-OK
OUTP      M02409	// IN-BUFF R-LD-OK 1P
; L75
LOAD      M02406	// IN-BUFF L-LD-OK
OR        M02408	// IN-BUFF R-LD-OK
OUT       M0240A	// LOAD-OK KP
// IN-BUFF CENTER  FPCB  ALIGN
; L78
LOAD NOT  M02407	// IN-BUFF L-LD-OK 1P
AND NOT   M02409	// IN-BUFF R-LD-OK 1P
AND NOT   M02430	// CENT ALIGN-CYC
AND NOT   M18633	// L-A©öAUTO AUAcAOA¨ö
AND NOT   M18643	// R-A©öAUTO AUAcAOA¨ö
NOT
LOAD NOT  M18202	// ¢¯¨­AE ¨ùO©ø¨£¡Æ¡§
AND NOT   M18204	// ¢¯A¢¬¡ÍAE ¨ùO©ø¨£¡Æ¡§
AND NOT   M18633	// L-A©öAUTO AUAcAOA¨ö
AND NOT   M18643	// R-A©öAUTO AUAcAOA¨ö
NOT
AND NOT   K00252	// LOADING ¡¾a ONLINE
OR LOAD
LOAD      T2001	// IN-BUFF RIGT(L-LD)
OR        T2000	// IN-BUFF LEFT(R-LD)
AND LOAD
LOAD NOT  M02435	// CENT FPCB ALIGN_ed
OR NOT    M02445	// IN-BUFF ALIGN_ed
AND LOAD
AND       M02412	// ANY AUTO-RUN
OUT       M02430	// CENT ALIGN-CYC

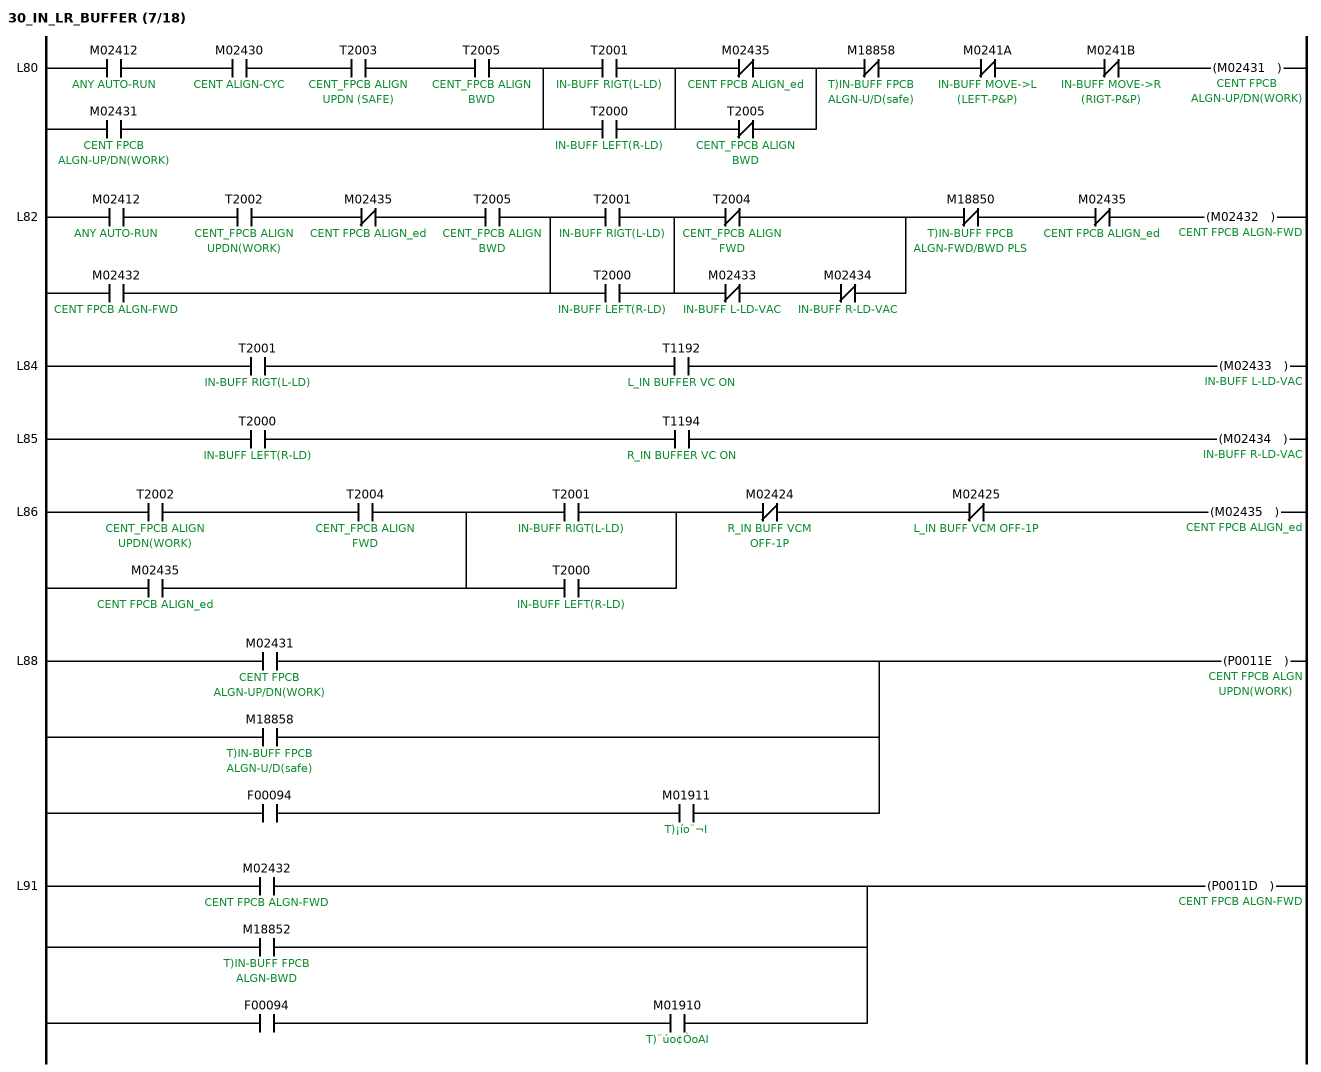
; L80
LOAD      M02412	// ANY AUTO-RUN
AND       M02430	// CENT ALIGN-CYC
AND       T2003	// CENT_FPCB ALIGN UPDN (SAFE)
AND       T2005	// CENT_FPCB ALIGN BWD
OR        M02431	// CENT FPCB ALGN-UP/DN(WORK)
LOAD      T2001	// IN-BUFF RIGT(L-LD)
OR        T2000	// IN-BUFF LEFT(R-LD)
AND LOAD
LOAD NOT  M02435	// CENT FPCB ALIGN_ed
OR NOT    T2005	// CENT_FPCB ALIGN BWD
AND LOAD
AND NOT   M18858	// T)IN-BUFF FPCB ALGN-U/D(safe)
AND NOT   M0241A	// IN-BUFF MOVE->L (LEFT-P&P)
AND NOT   M0241B	// IN-BUFF MOVE->R (RIGT-P&P)
OUT       M02431	// CENT FPCB ALGN-UP/DN(WORK)
; L82
LOAD      M02412	// ANY AUTO-RUN
AND       T2002	// CENT_FPCB ALIGN UPDN(WORK)
AND NOT   M02435	// CENT FPCB ALIGN_ed
AND       T2005	// CENT_FPCB ALIGN BWD
OR        M02432	// CENT FPCB ALGN-FWD
LOAD      T2001	// IN-BUFF RIGT(L-LD)
OR        T2000	// IN-BUFF LEFT(R-LD)
AND LOAD
LOAD NOT  T2004	// CENT_FPCB ALIGN FWD
LOAD NOT  M02433	// IN-BUFF L-LD-VAC
AND NOT   M02434	// IN-BUFF R-LD-VAC
OR LOAD
AND LOAD
AND NOT   M18850	// T)IN-BUFF FPCB ALGN-FWD/BWD PLS
AND NOT   M02435	// CENT FPCB ALIGN_ed
OUT       M02432	// CENT FPCB ALGN-FWD
; L84
LOAD      T2001	// IN-BUFF RIGT(L-LD)
AND       T1192	// L_IN BUFFER VC ON
OUT       M02433	// IN-BUFF L-LD-VAC
; L85
LOAD      T2000	// IN-BUFF LEFT(R-LD)
AND       T1194	// R_IN BUFFER VC ON
OUT       M02434	// IN-BUFF R-LD-VAC
; L86
LOAD      T2002	// CENT_FPCB ALIGN UPDN(WORK)
AND       T2004	// CENT_FPCB ALIGN FWD
OR        M02435	// CENT FPCB ALIGN_ed
LOAD      T2001	// IN-BUFF RIGT(L-LD)
OR        T2000	// IN-BUFF LEFT(R-LD)
AND LOAD
AND NOT   M02424	// R_IN BUFF VCM OFF-1P
AND NOT   M02425	// L_IN BUFF VCM OFF-1P
OUT       M02435	// CENT FPCB ALIGN_ed
; L88
LOAD      M02431	// CENT FPCB ALGN-UP/DN(WORK)
OR        M18858	// T)IN-BUFF FPCB ALGN-U/D(safe)
LOAD      F00094
AND       M01911	// T)¡ío¨¬I
OR LOAD
OUT       P0011E	// CENT FPCB ALGN UPDN(WORK)
; L91
LOAD      M02432	// CENT FPCB ALGN-FWD
OR        M18852	// T)IN-BUFF FPCB ALGN-BWD
LOAD      F00094
AND       M01910	// T)¨úo¢ÒoAI
OR LOAD
OUT       P0011D	// CENT FPCB ALGN-FWD

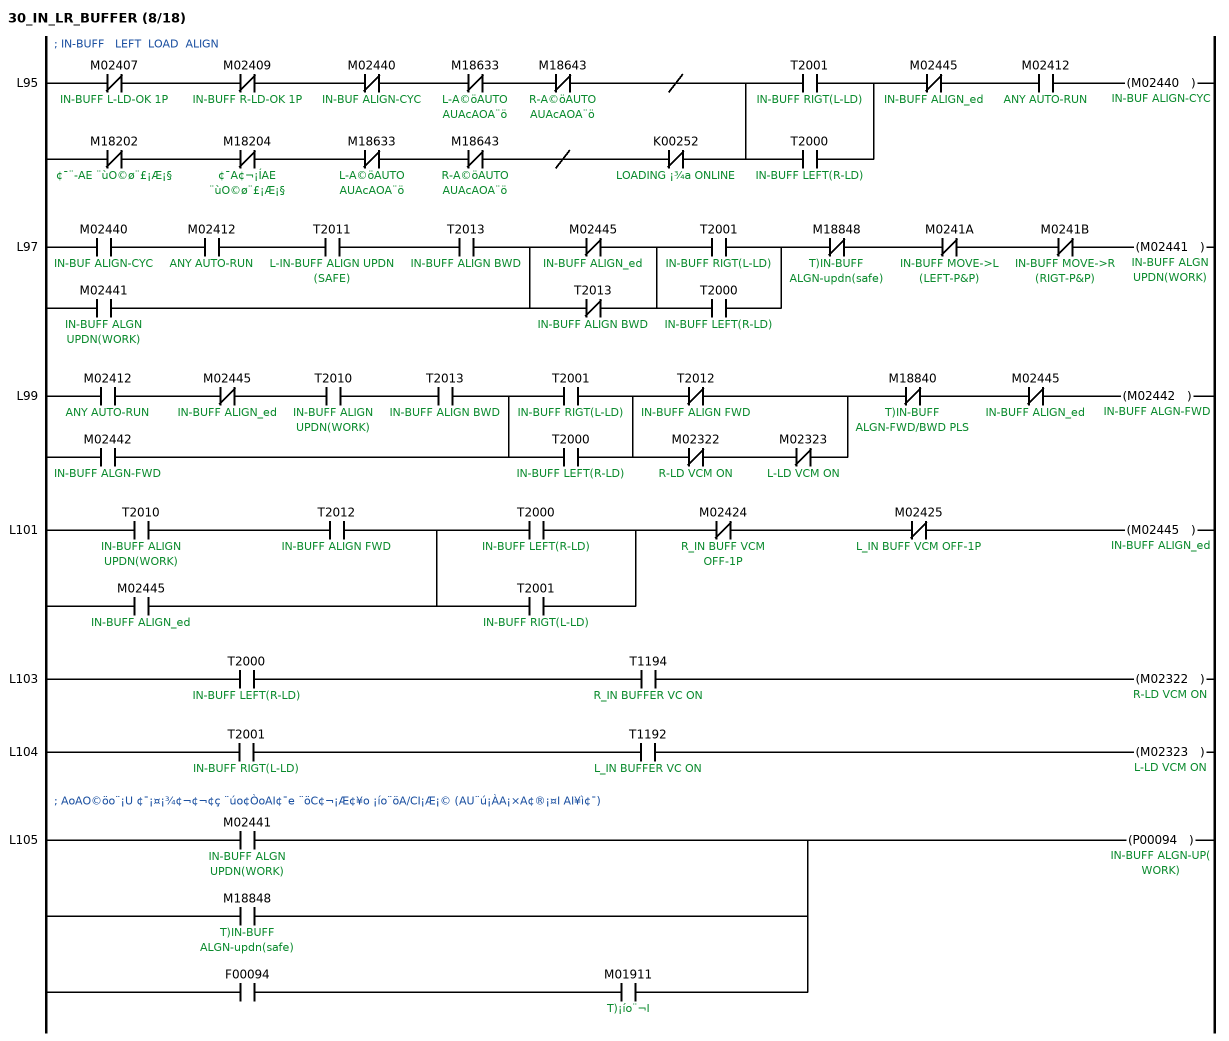
// IN-BUFF   LEFT  LOAD  ALIGN
; L95
LOAD NOT  M02407	// IN-BUFF L-LD-OK 1P
AND NOT   M02409	// IN-BUFF R-LD-OK 1P
AND NOT   M02440	// IN-BUF ALIGN-CYC
AND NOT   M18633	// L-A©öAUTO AUAcAOA¨ö
AND NOT   M18643	// R-A©öAUTO AUAcAOA¨ö
NOT
LOAD NOT  M18202	// ¢¯¨­AE ¨ùO©ø¨£¡Æ¡§
AND NOT   M18204	// ¢¯A¢¬¡ÍAE ¨ùO©ø¨£¡Æ¡§
AND NOT   M18633	// L-A©öAUTO AUAcAOA¨ö
AND NOT   M18643	// R-A©öAUTO AUAcAOA¨ö
NOT
AND NOT   K00252	// LOADING ¡¾a ONLINE
OR LOAD
LOAD      T2001	// IN-BUFF RIGT(L-LD)
OR        T2000	// IN-BUFF LEFT(R-LD)
AND LOAD
AND NOT   M02445	// IN-BUFF ALIGN_ed
AND       M02412	// ANY AUTO-RUN
OUT       M02440	// IN-BUF ALIGN-CYC
; L97
LOAD      M02440	// IN-BUF ALIGN-CYC
AND       M02412	// ANY AUTO-RUN
AND       T2011	// L-IN-BUFF ALIGN UPDN (SAFE)
AND       T2013	// IN-BUFF ALIGN BWD
OR        M02441	// IN-BUFF ALGN UPDN(WORK)
LOAD NOT  M02445	// IN-BUFF ALIGN_ed
OR NOT    T2013	// IN-BUFF ALIGN BWD
AND LOAD
LOAD      T2001	// IN-BUFF RIGT(L-LD)
OR        T2000	// IN-BUFF LEFT(R-LD)
AND LOAD
AND NOT   M18848	// T)IN-BUFF ALGN-updn(safe)
AND NOT   M0241A	// IN-BUFF MOVE->L (LEFT-P&P)
AND NOT   M0241B	// IN-BUFF MOVE->R (RIGT-P&P)
OUT       M02441	// IN-BUFF ALGN UPDN(WORK)
; L99
LOAD      M02412	// ANY AUTO-RUN
AND NOT   M02445	// IN-BUFF ALIGN_ed
AND       T2010	// IN-BUFF ALIGN UPDN(WORK)
AND       T2013	// IN-BUFF ALIGN BWD
OR        M02442	// IN-BUFF ALGN-FWD
LOAD      T2001	// IN-BUFF RIGT(L-LD)
OR        T2000	// IN-BUFF LEFT(R-LD)
AND LOAD
LOAD NOT  T2012	// IN-BUFF ALIGN FWD
LOAD NOT  M02322	// R-LD VCM ON
AND NOT   M02323	// L-LD VCM ON
OR LOAD
AND LOAD
AND NOT   M18840	// T)IN-BUFF ALGN-FWD/BWD PLS
AND NOT   M02445	// IN-BUFF ALIGN_ed
OUT       M02442	// IN-BUFF ALGN-FWD
; L101
LOAD      T2010	// IN-BUFF ALIGN UPDN(WORK)
AND       T2012	// IN-BUFF ALIGN FWD
OR        M02445	// IN-BUFF ALIGN_ed
LOAD      T2000	// IN-BUFF LEFT(R-LD)
OR        T2001	// IN-BUFF RIGT(L-LD)
AND LOAD
AND NOT   M02424	// R_IN BUFF VCM OFF-1P
AND NOT   M02425	// L_IN BUFF VCM OFF-1P
OUT       M02445	// IN-BUFF ALIGN_ed
; L103
LOAD      T2000	// IN-BUFF LEFT(R-LD)
AND       T1194	// R_IN BUFFER VC ON
OUT       M02322	// R-LD VCM ON
; L104
LOAD      T2001	// IN-BUFF RIGT(L-LD)
AND       T1192	// L_IN BUFFER VC ON
OUT       M02323	// L-LD VCM ON
; L105
LOAD      M02441	// IN-BUFF ALGN UPDN(WORK)
OR        M18848	// T)IN-BUFF ALGN-updn(safe)
LOAD      F00094
AND       M01911	// T)¡ío¨¬I
OR LOAD
OUT       P00094	// IN-BUFF ALGN-UP(WORK)
// output comment: AoAO©öo¨¡U ¢¯¡¤¡¾¢¬¢¬¢ç ¨úo¢ÒoAI¢¯e ¨öC¢¬¡Æ¢¥o ¡ío¨öA/CI¡Æ¡© (AU¨ú¡ÀA¡×A¢®¡¤I AI¥ì¢¯)

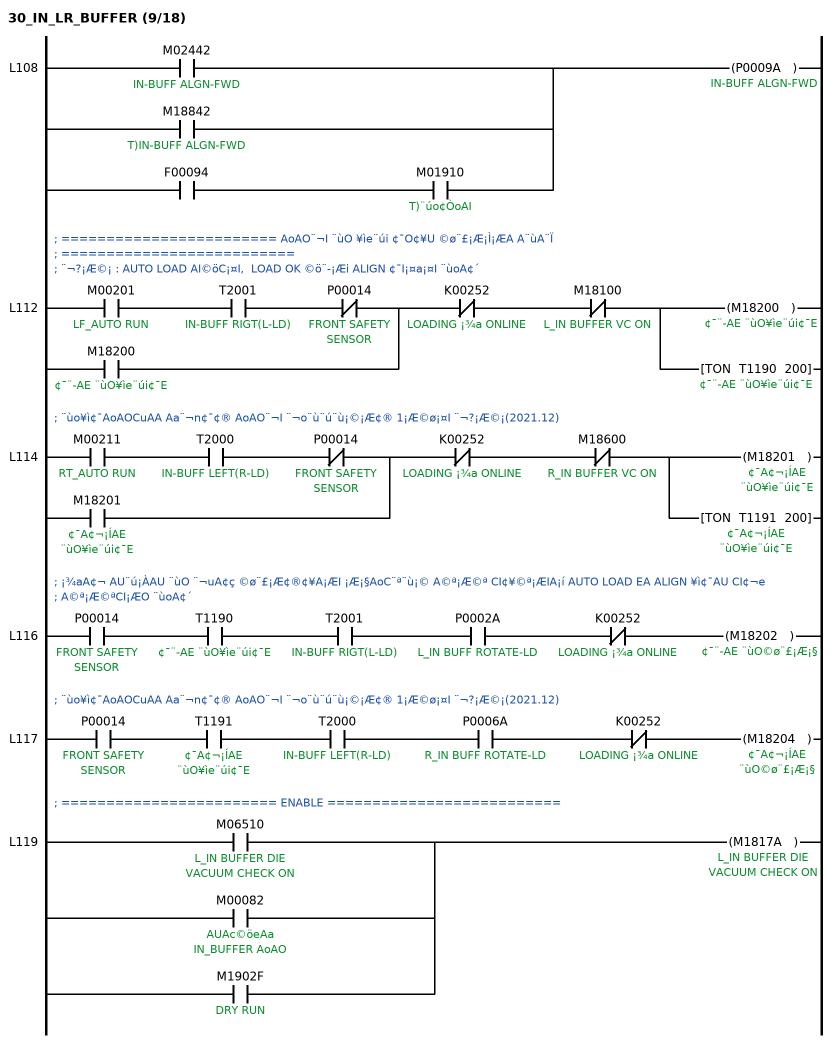
; L108
LOAD      M02442	// IN-BUFF ALGN-FWD
OR        M18842	// T)IN-BUFF ALGN-FWD
LOAD      F00094
AND       M01910	// T)¨úo¢ÒoAI
OR LOAD
OUT       P0009A	// IN-BUFF ALGN-FWD
// ======================== AoAO¨¬I ¨ùO ¥ìe¨úi ¢¯O¢¥U ©ø¨£¡Æ¡Ì¡ÆA A¨ùA¨Ï ==========================
// 
// ¨¬?¡Æ©¡ : AUTO LOAD AI©öC¡¤I,  LOAD OK ©ö¨­¡Æi ALIGN ¢¯I¡¤a¡¤I ¨ùoA¢´
; L112
LOAD      M00201	// LF_AUTO RUN
AND       T2001	// IN-BUFF RIGT(L-LD)
AND NOT   P00014	// FRONT SAFETY SENSOR
OR        M18200	// ¢¯¨­AE ¨ùO¥ìe¨úi¢¯E
AND NOT   K00252	// LOADING ¡¾a ONLINE
AND NOT   M18100	// L_IN BUFFER VC ON
OUT       M18200	// ¢¯¨­AE ¨ùO¥ìe¨úi¢¯E
TON       T1190 200	// ¢¯¨­AE ¨ùO¥ìe¨úi¢¯E
; L114
LOAD      M00211	// RT_AUTO RUN
AND       T2000	// IN-BUFF LEFT(R-LD)
AND NOT   P00014	// FRONT SAFETY SENSOR
OR        M18201	// ¢¯A¢¬¡ÍAE ¨ùO¥ìe¨úi¢¯E
AND NOT   K00252	// LOADING ¡¾a ONLINE
AND NOT   M18600	// R_IN BUFFER VC ON
OUT       M18201	// ¢¯A¢¬¡ÍAE ¨ùO¥ìe¨úi¢¯E
TON       T1191 200	// ¢¯A¢¬¡ÍAE ¨ùO¥ìe¨úi¢¯E
// output comment: ¨ùo¥ì¢¯AoAOCuAA Aa¨¬n¢¯¢® AoAO¨¬I ¨¬o¨ù¨ú¨ù¡©¡Æ¢® 1¡Æ©ø¡¤I ¨¬?¡Æ©¡(2021.12)
; L116
LOAD      P00014	// FRONT SAFETY SENSOR
AND       T1190	// ¢¯¨­AE ¨ùO¥ìe¨úi¢¯E
AND       T2001	// IN-BUFF RIGT(L-LD)
AND       P0002A	// L_IN BUFF ROTATE-LD
AND NOT   K00252	// LOADING ¡¾a ONLINE
OUT       M18202	// ¢¯¨­AE ¨ùO©ø¨£¡Æ¡§
// output comment: ¡¾aA¢¬ AU¨ú¡ÀAU ¨ùO ¨¬uA¢ç ©ø¨£¡Æ¢®¢¥A¡ÆI ¡Æ¡§AoC¨ª¨ù¡© A©ª¡Æ©ª CI¢¥©ª¡ÆIA¡í AUTO LOAD EA ALIGN ¥ì¢¯AU CI¢¬e A©ª¡Æ©ªCI¡ÆO ¨ùoA¢´
; L117
LOAD      P00014	// FRONT SAFETY SENSOR
AND       T1191	// ¢¯A¢¬¡ÍAE ¨ùO¥ìe¨úi¢¯E
AND       T2000	// IN-BUFF LEFT(R-LD)
AND       P0006A	// R_IN BUFF ROTATE-LD
AND NOT   K00252	// LOADING ¡¾a ONLINE
OUT       M18204	// ¢¯A¢¬¡ÍAE ¨ùO©ø¨£¡Æ¡§
// output comment: ¨ùo¥ì¢¯AoAOCuAA Aa¨¬n¢¯¢® AoAO¨¬I ¨¬o¨ù¨ú¨ù¡©¡Æ¢® 1¡Æ©ø¡¤I ¨¬?¡Æ©¡(2021.12)
// ======================== ENABLE ==========================
; L119
LOAD      M06510	// L_IN BUFFER DIE VACUUM CHECK ON
OR        M00082	// AUAc©öeAa IN_BUFFER AoAO 
OR        M1902F	// DRY RUN
OUT       M1817A	// L_IN BUFFER DIE VACUUM CHECK ON

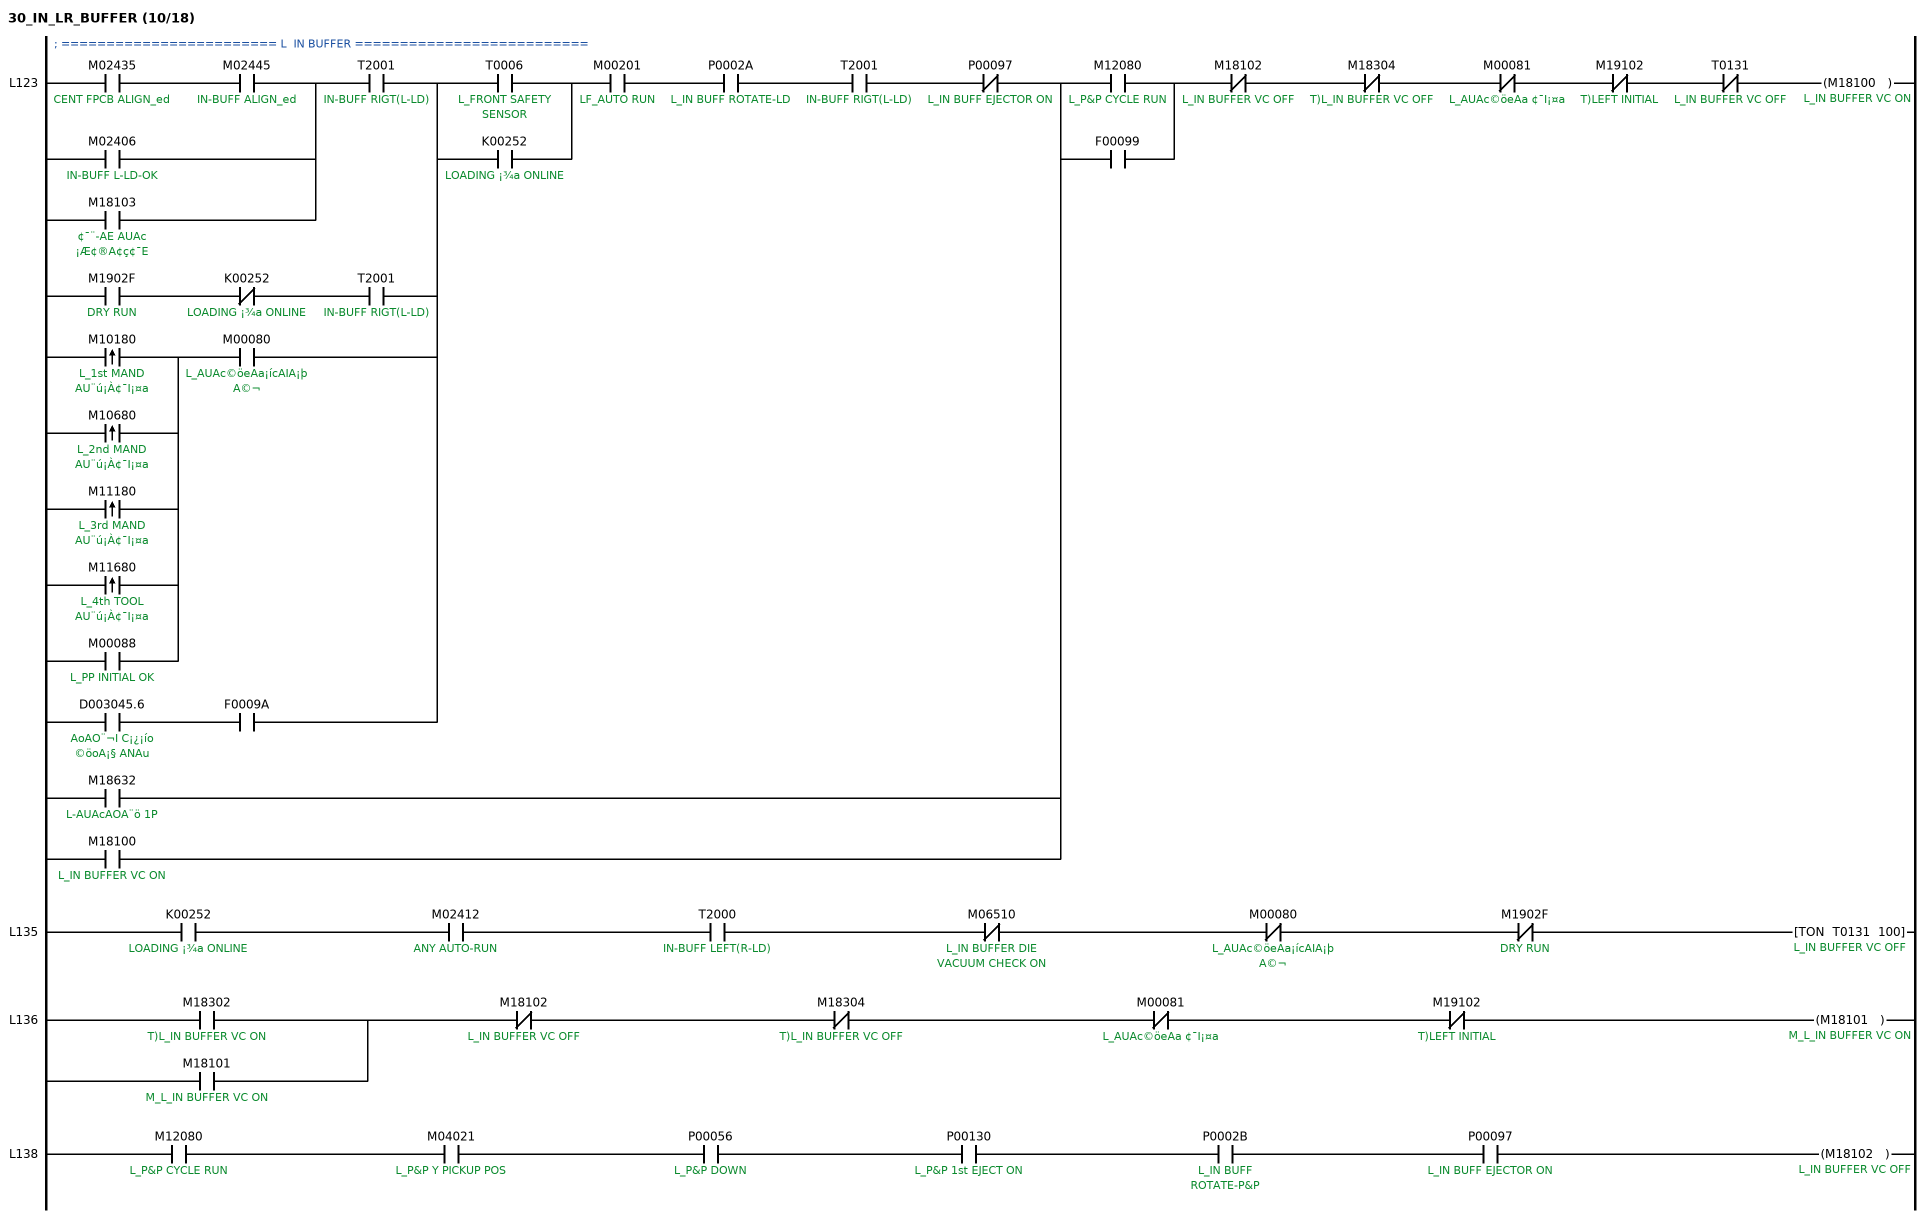
// ======================== L  IN BUFFER ==========================
; L123
LOAD      M02435	// CENT FPCB ALIGN_ed
AND       M02445	// IN-BUFF ALIGN_ed
OR        M02406	// IN-BUFF L-LD-OK
OR        M18103	// ¢¯¨­AE AUAc ¡Æ¢®A¢ç¢¯E
AND       T2001	// IN-BUFF RIGT(L-LD)
LOAD      M1902F	// DRY RUN
AND NOT   K00252	// LOADING ¡¾a ONLINE
AND       T2001	// IN-BUFF RIGT(L-LD)
OR LOAD
LOADP     M10180	// L_1st MAND AU¨ú¡À¢¯I¡¤a
ORP       M10680	// L_2nd MAND AU¨ú¡À¢¯I¡¤a
ORP       M11180	// L_3rd MAND AU¨ú¡À¢¯I¡¤a
ORP       M11680	// L_4th TOOL AU¨ú¡À¢¯I¡¤a
OR        M00088	// L_PP INITIAL OK
AND       M00080	// L_AUAc©öeAa¡ícAIA¡þA©¬
OR LOAD
LOAD      D003045.6	// AoAO¨¬I C¡¿¡ío ©öoA¡§ ANAu
AND       F0009A
OR LOAD
LOAD      T0006	// L_FRONT SAFETY SENSOR
OR        K00252	// LOADING ¡¾a ONLINE
AND LOAD
AND       M00201	// LF_AUTO RUN
AND       P0002A	// L_IN BUFF ROTATE-LD
AND       T2001	// IN-BUFF RIGT(L-LD)
AND NOT   P00097	// L_IN BUFF EJECTOR ON
OR        M18632	// L-AUAcAOA¨ö 1P
OR        M18100	// L_IN BUFFER VC ON
LOAD      M12080	// L_P&P CYCLE RUN
OR        F00099
AND LOAD
AND NOT   M18102	// L_IN BUFFER VC OFF
AND NOT   M18304	// T)L_IN BUFFER VC OFF
AND NOT   M00081	// L_AUAc©öeAa ¢¯I¡¤a
AND NOT   M19102	// T)LEFT INITIAL
AND NOT   T0131	// L_IN BUFFER VC OFF
OUT       M18100	// L_IN BUFFER VC ON
; L135
LOAD      K00252	// LOADING ¡¾a ONLINE
AND       M02412	// ANY AUTO-RUN
AND       T2000	// IN-BUFF LEFT(R-LD)
AND NOT   M06510	// L_IN BUFFER DIE VACUUM CHECK ON
AND NOT   M00080	// L_AUAc©öeAa¡ícAIA¡þA©¬
AND NOT   M1902F	// DRY RUN
TON       T0131 100	// L_IN BUFFER VC OFF
; L136
LOAD      M18302	// T)L_IN BUFFER VC ON
OR        M18101	// M_L_IN BUFFER VC ON
AND NOT   M18102	// L_IN BUFFER VC OFF
AND NOT   M18304	// T)L_IN BUFFER VC OFF
AND NOT   M00081	// L_AUAc©öeAa ¢¯I¡¤a
AND NOT   M19102	// T)LEFT INITIAL
OUT       M18101	// M_L_IN BUFFER VC ON
; L138
LOAD      M12080	// L_P&P CYCLE RUN
AND       M04021	// L_P&P Y PICKUP POS
AND       P00056	// L_P&P DOWN
AND       P00130	// L_P&P 1st EJECT ON
AND       P0002B	// L_IN BUFF ROTATE-P&P
AND       P00097	// L_IN BUFF EJECTOR ON
OUT       M18102	// L_IN BUFFER VC OFF

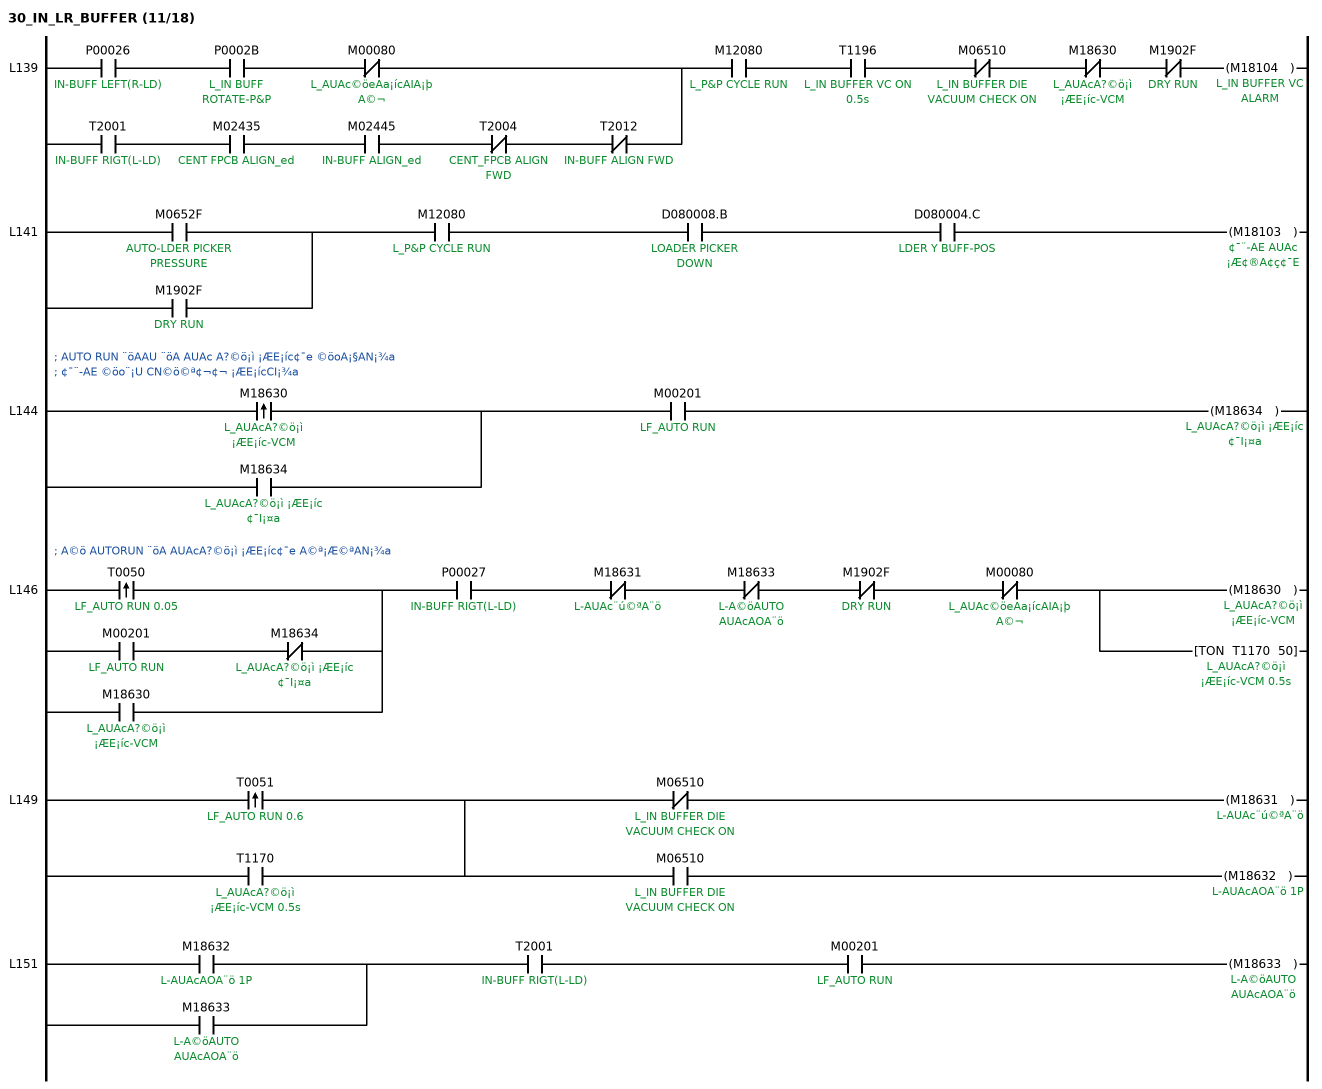
; L139
LOAD      P00026	// IN-BUFF LEFT(R-LD)
AND       P0002B	// L_IN BUFF ROTATE-P&P
AND NOT   M00080	// L_AUAc©öeAa¡ícAIA¡þA©¬
LOAD      T2001	// IN-BUFF RIGT(L-LD)
AND       M02435	// CENT FPCB ALIGN_ed
AND       M02445	// IN-BUFF ALIGN_ed
AND NOT   T2004	// CENT_FPCB ALIGN FWD
AND NOT   T2012	// IN-BUFF ALIGN FWD
OR LOAD
AND       M12080	// L_P&P CYCLE RUN
AND       T1196	// L_IN BUFFER VC ON 0.5s
AND NOT   M06510	// L_IN BUFFER DIE VACUUM CHECK ON
AND NOT   M18630	// L_AUAcA?©ö¡ì ¡ÆE¡íc-VCM
AND NOT   M1902F	// DRY RUN
OUT       M18104	// L_IN BUFFER VC ALARM
; L141
LOAD      M0652F	// AUTO-LDER PICKER PRESSURE
OR        M1902F	// DRY RUN
AND       M12080	// L_P&P CYCLE RUN
AND       D080008.B	// LOADER PICKER DOWN
AND       D080004.C	// LDER Y BUFF-POS
OUT       M18103	// ¢¯¨­AE AUAc ¡Æ¢®A¢ç¢¯E
// AUTO RUN ¨öAAU ¨öA AUAc A?©ö¡ì ¡ÆE¡íc¢¯e ©öoA¡§AN¡¾a
; L144
LOADP     M18630	// L_AUAcA?©ö¡ì ¡ÆE¡íc-VCM
OR        M18634	// L_AUAcA?©ö¡ì ¡ÆE¡íc ¢¯I¡¤a
AND       M00201	// LF_AUTO RUN
OUT       M18634	// L_AUAcA?©ö¡ì ¡ÆE¡íc ¢¯I¡¤a
// output comment: ¢¯¨­AE ©öo¨¡U CN©ö©ª¢¬¢¬ ¡ÆE¡ícCI¡¾a
; L146
LOADP     T0050	// LF_AUTO RUN 0.05
LOAD      M00201	// LF_AUTO RUN
AND NOT   M18634	// L_AUAcA?©ö¡ì ¡ÆE¡íc ¢¯I¡¤a
OR LOAD
OR        M18630	// L_AUAcA?©ö¡ì ¡ÆE¡íc-VCM
AND       P00027	// IN-BUFF RIGT(L-LD)
AND NOT   M18631	// L-AUAc¨ú©ªA¨ö
AND NOT   M18633	// L-A©öAUTO AUAcAOA¨ö
AND NOT   M1902F	// DRY RUN
AND NOT   M00080	// L_AUAc©öeAa¡ícAIA¡þA©¬
OUT       M18630	// L_AUAcA?©ö¡ì ¡ÆE¡íc-VCM
TON       T1170 50	// L_AUAcA?©ö¡ì ¡ÆE¡íc-VCM 0.5s
// output comment: A©ö AUTORUN ¨öA AUAcA?©ö¡ì ¡ÆE¡íc¢¯e A©ª¡Æ©ªAN¡¾a
; L149
LOADP     T0051	// LF_AUTO RUN 0.6
OR        T1170	// L_AUAcA?©ö¡ì ¡ÆE¡íc-VCM 0.5s
MPUSH
AND NOT   M06510	// L_IN BUFFER DIE VACUUM CHECK ON
OUT       M18631	// L-AUAc¨ú©ªA¨ö
MPOP
AND       M06510	// L_IN BUFFER DIE VACUUM CHECK ON
OUT       M18632	// L-AUAcAOA¨ö 1P
; L151
LOAD      M18632	// L-AUAcAOA¨ö 1P
OR        M18633	// L-A©öAUTO AUAcAOA¨ö
AND       T2001	// IN-BUFF RIGT(L-LD)
AND       M00201	// LF_AUTO RUN
OUT       M18633	// L-A©öAUTO AUAcAOA¨ö

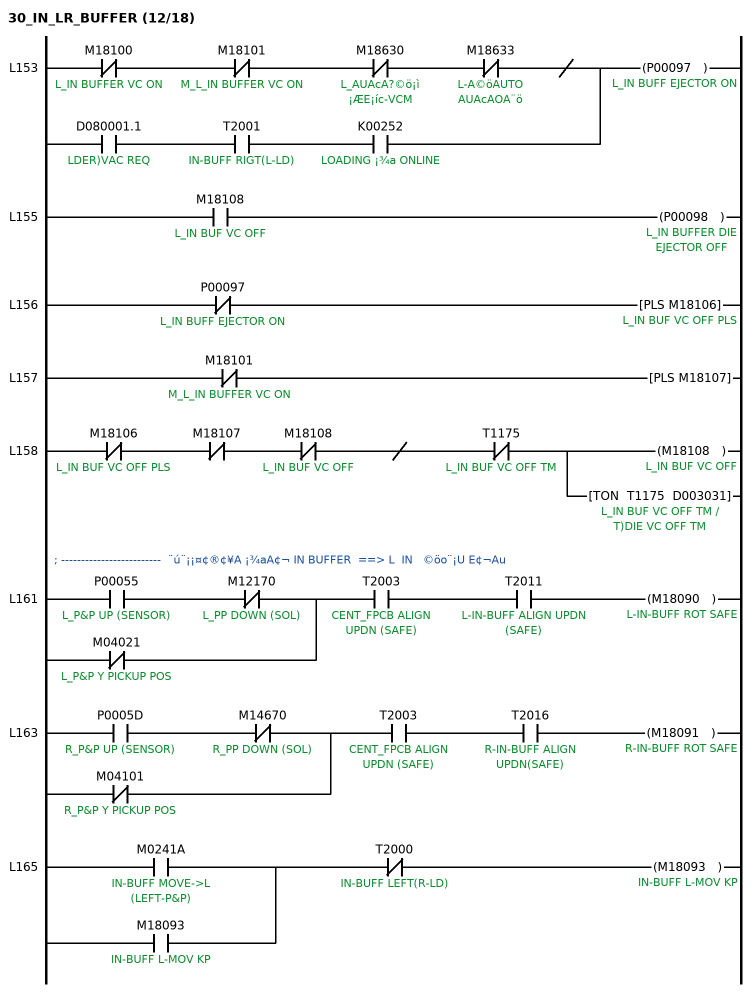
; L153
LOAD NOT  M18100	// L_IN BUFFER VC ON
AND NOT   M18101	// M_L_IN BUFFER VC ON
AND NOT   M18630	// L_AUAcA?©ö¡ì ¡ÆE¡íc-VCM
AND NOT   M18633	// L-A©öAUTO AUAcAOA¨ö
NOT
LOAD      D080001.1	// LDER)VAC REQ
AND       T2001	// IN-BUFF RIGT(L-LD)
AND       K00252	// LOADING ¡¾a ONLINE
OR LOAD
OUT       P00097	// L_IN BUFF EJECTOR ON
; L155
LOAD      M18108	// L_IN BUF VC OFF
OUT       P00098	// L_IN BUFFER DIE EJECTOR OFF
; L156
LOAD NOT  P00097	// L_IN BUFF EJECTOR ON
OUTP      M18106	// L_IN BUF VC OFF PLS
; L157
LOAD NOT  M18101	// M_L_IN BUFFER VC ON
OUTP      M18107
; L158
LOAD NOT  M18106	// L_IN BUF VC OFF PLS
AND NOT   M18107
AND NOT   M18108	// L_IN BUF VC OFF
NOT
AND NOT   T1175	// L_IN BUF VC OFF TM
OUT       M18108	// L_IN BUF VC OFF
TON       T1175 D003031	// L_IN BUF VC OFF TM / T)DIE VC OFF TM
// -------------------------  ¨ú¨¡¡¤¢®¢¥A ¡¾aA¢¬ IN BUFFER  ==> L  IN   ©öo¨¡U E¢¬Au
; L161
LOAD      P00055	// L_P&P UP (SENSOR)
AND NOT   M12170	// L_PP DOWN (SOL)
OR NOT    M04021	// L_P&P Y PICKUP POS
AND       T2003	// CENT_FPCB ALIGN UPDN (SAFE)
AND       T2011	// L-IN-BUFF ALIGN UPDN (SAFE)
OUT       M18090	// L-IN-BUFF ROT SAFE
; L163
LOAD      P0005D	// R_P&P UP (SENSOR)
AND NOT   M14670	// R_PP DOWN (SOL)
OR NOT    M04101	// R_P&P Y PICKUP POS
AND       T2003	// CENT_FPCB ALIGN UPDN (SAFE)
AND       T2016	// R-IN-BUFF ALIGN UPDN(SAFE)
OUT       M18091	// R-IN-BUFF ROT SAFE
; L165
LOAD      M0241A	// IN-BUFF MOVE->L (LEFT-P&P)
OR        M18093	// IN-BUFF L-MOV KP
AND NOT   T2000	// IN-BUFF LEFT(R-LD)
OUT       M18093	// IN-BUFF L-MOV KP

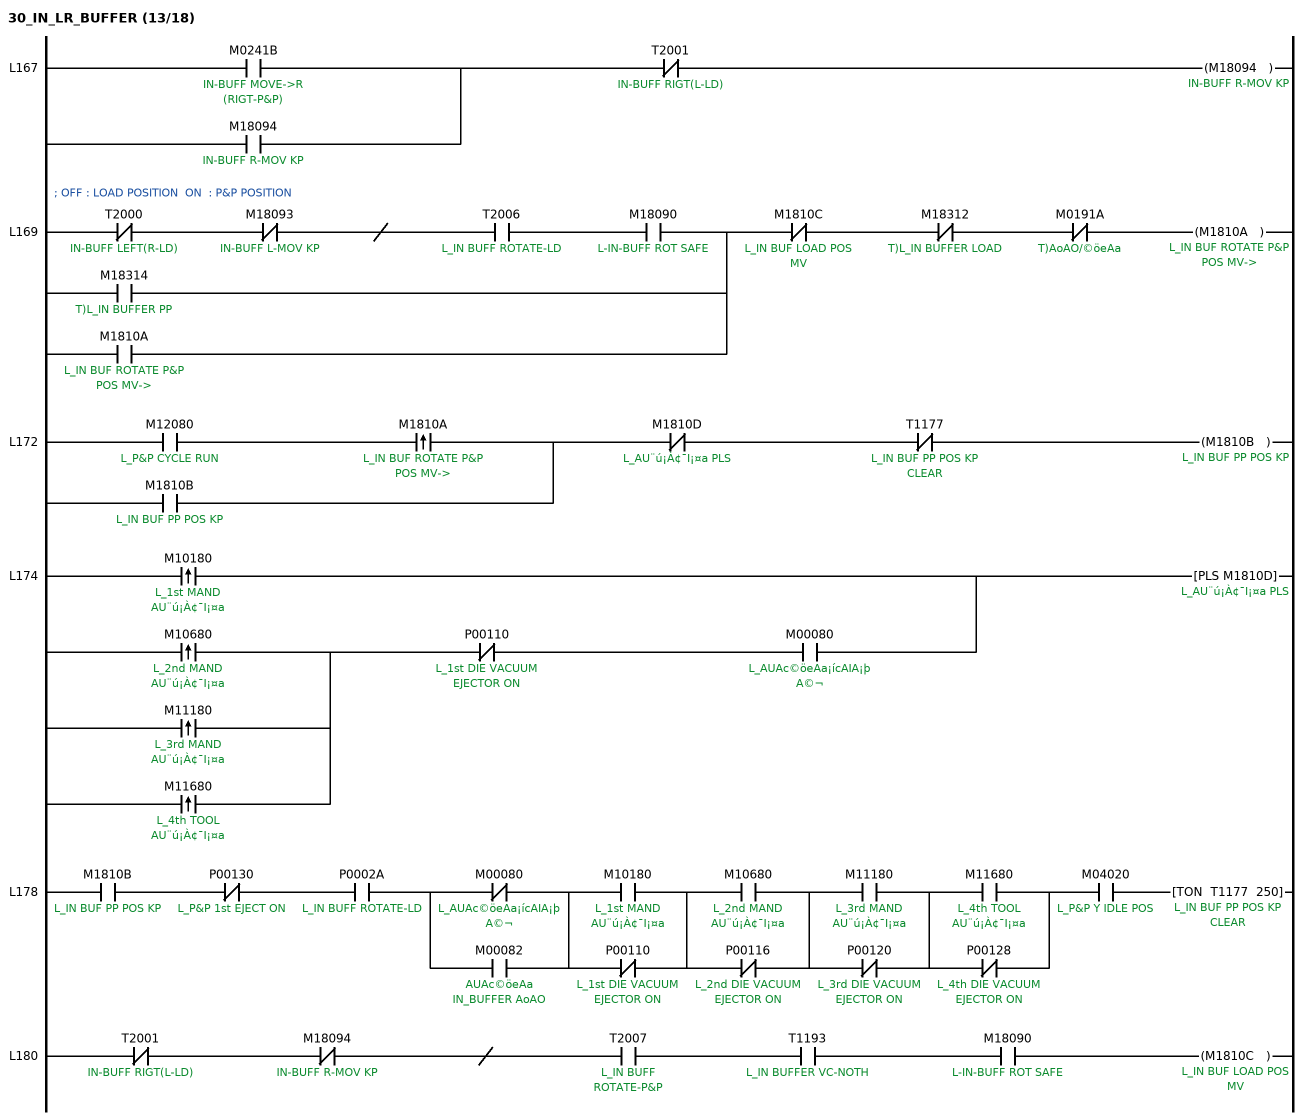
; L167
LOAD      M0241B	// IN-BUFF MOVE->R (RIGT-P&P)
OR        M18094	// IN-BUFF R-MOV KP
AND NOT   T2001	// IN-BUFF RIGT(L-LD)
OUT       M18094	// IN-BUFF R-MOV KP
; L169
LOAD NOT  T2000	// IN-BUFF LEFT(R-LD)
AND NOT   M18093	// IN-BUFF L-MOV KP
NOT
AND       T2006	// L_IN BUFF ROTATE-LD
AND       M18090	// L-IN-BUFF ROT SAFE
OR        M18314	// T)L_IN BUFFER PP
OR        M1810A	// L_IN BUF ROTATE P&P POS MV->
AND NOT   M1810C	// L_IN BUF LOAD POS MV
AND NOT   M18312	// T)L_IN BUFFER LOAD
AND NOT   M0191A	// T)AoAO/©öeAa
OUT       M1810A	// L_IN BUF ROTATE P&P POS MV->
// output comment: OFF : LOAD POSITION  ON  : P&P POSITION
; L172
LOAD      M12080	// L_P&P CYCLE RUN
ANDP      M1810A	// L_IN BUF ROTATE P&P POS MV->
OR        M1810B	// L_IN BUF PP POS KP
AND NOT   M1810D	// L_AU¨ú¡À¢¯I¡¤a PLS
AND NOT   T1177	// L_IN BUF PP POS KP CLEAR
OUT       M1810B	// L_IN BUF PP POS KP
; L174
LOADP     M10180	// L_1st MAND AU¨ú¡À¢¯I¡¤a
LOADP     M10680	// L_2nd MAND AU¨ú¡À¢¯I¡¤a
ORP       M11180	// L_3rd MAND AU¨ú¡À¢¯I¡¤a
ORP       M11680	// L_4th TOOL AU¨ú¡À¢¯I¡¤a
AND NOT   P00110	// L_1st DIE VACUUM EJECTOR ON
AND       M00080	// L_AUAc©öeAa¡ícAIA¡þA©¬
OR LOAD
OUTP      M1810D	// L_AU¨ú¡À¢¯I¡¤a PLS
; L178
LOAD      M1810B	// L_IN BUF PP POS KP
AND NOT   P00130	// L_P&P 1st EJECT ON
AND       P0002A	// L_IN BUFF ROTATE-LD
LOAD NOT  M00080	// L_AUAc©öeAa¡ícAIA¡þA©¬
OR        M00082	// AUAc©öeAa IN_BUFFER AoAO 
AND LOAD
LOAD      M10180	// L_1st MAND AU¨ú¡À¢¯I¡¤a
OR NOT    P00110	// L_1st DIE VACUUM EJECTOR ON
AND LOAD
LOAD      M10680	// L_2nd MAND AU¨ú¡À¢¯I¡¤a
OR NOT    P00116	// L_2nd DIE VACUUM EJECTOR ON
AND LOAD
LOAD      M11180	// L_3rd MAND AU¨ú¡À¢¯I¡¤a
OR NOT    P00120	// L_3rd DIE VACUUM EJECTOR ON
AND LOAD
LOAD      M11680	// L_4th TOOL AU¨ú¡À¢¯I¡¤a
OR NOT    P00128	// L_4th DIE VACUUM EJECTOR ON
AND LOAD
AND       M04020	// L_P&P Y IDLE POS
TON       T1177 250	// L_IN BUF PP POS KP CLEAR
; L180
LOAD NOT  T2001	// IN-BUFF RIGT(L-LD)
AND NOT   M18094	// IN-BUFF R-MOV KP
NOT
AND       T2007	// L_IN BUFF ROTATE-P&P
AND       T1193	// L_IN BUFFER VC-NOTH
AND       M18090	// L-IN-BUFF ROT SAFE
OUT       M1810C	// L_IN BUF LOAD POS MV

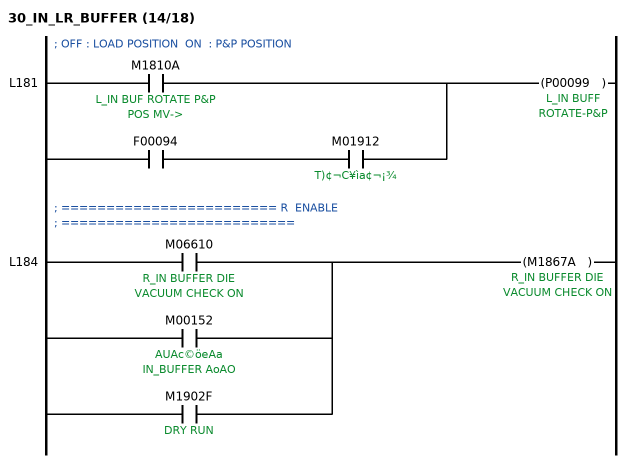
; L181
LOAD      M1810A	// L_IN BUF ROTATE P&P POS MV->
LOAD      F00094
AND       M01912	// T)¢¬C¥ìa¢¬¡¾
OR LOAD
OUT       P00099	// L_IN BUFF ROTATE-P&P
// output comment: OFF : LOAD POSITION  ON  : P&P POSITION
// ======================== R  ENABLE ==========================
; L184
LOAD      M06610	// R_IN BUFFER DIE VACUUM CHECK ON
OR        M00152	// AUAc©öeAa IN_BUFFER AoAO 
OR        M1902F	// DRY RUN
OUT       M1867A	// R_IN BUFFER DIE VACUUM CHECK ON

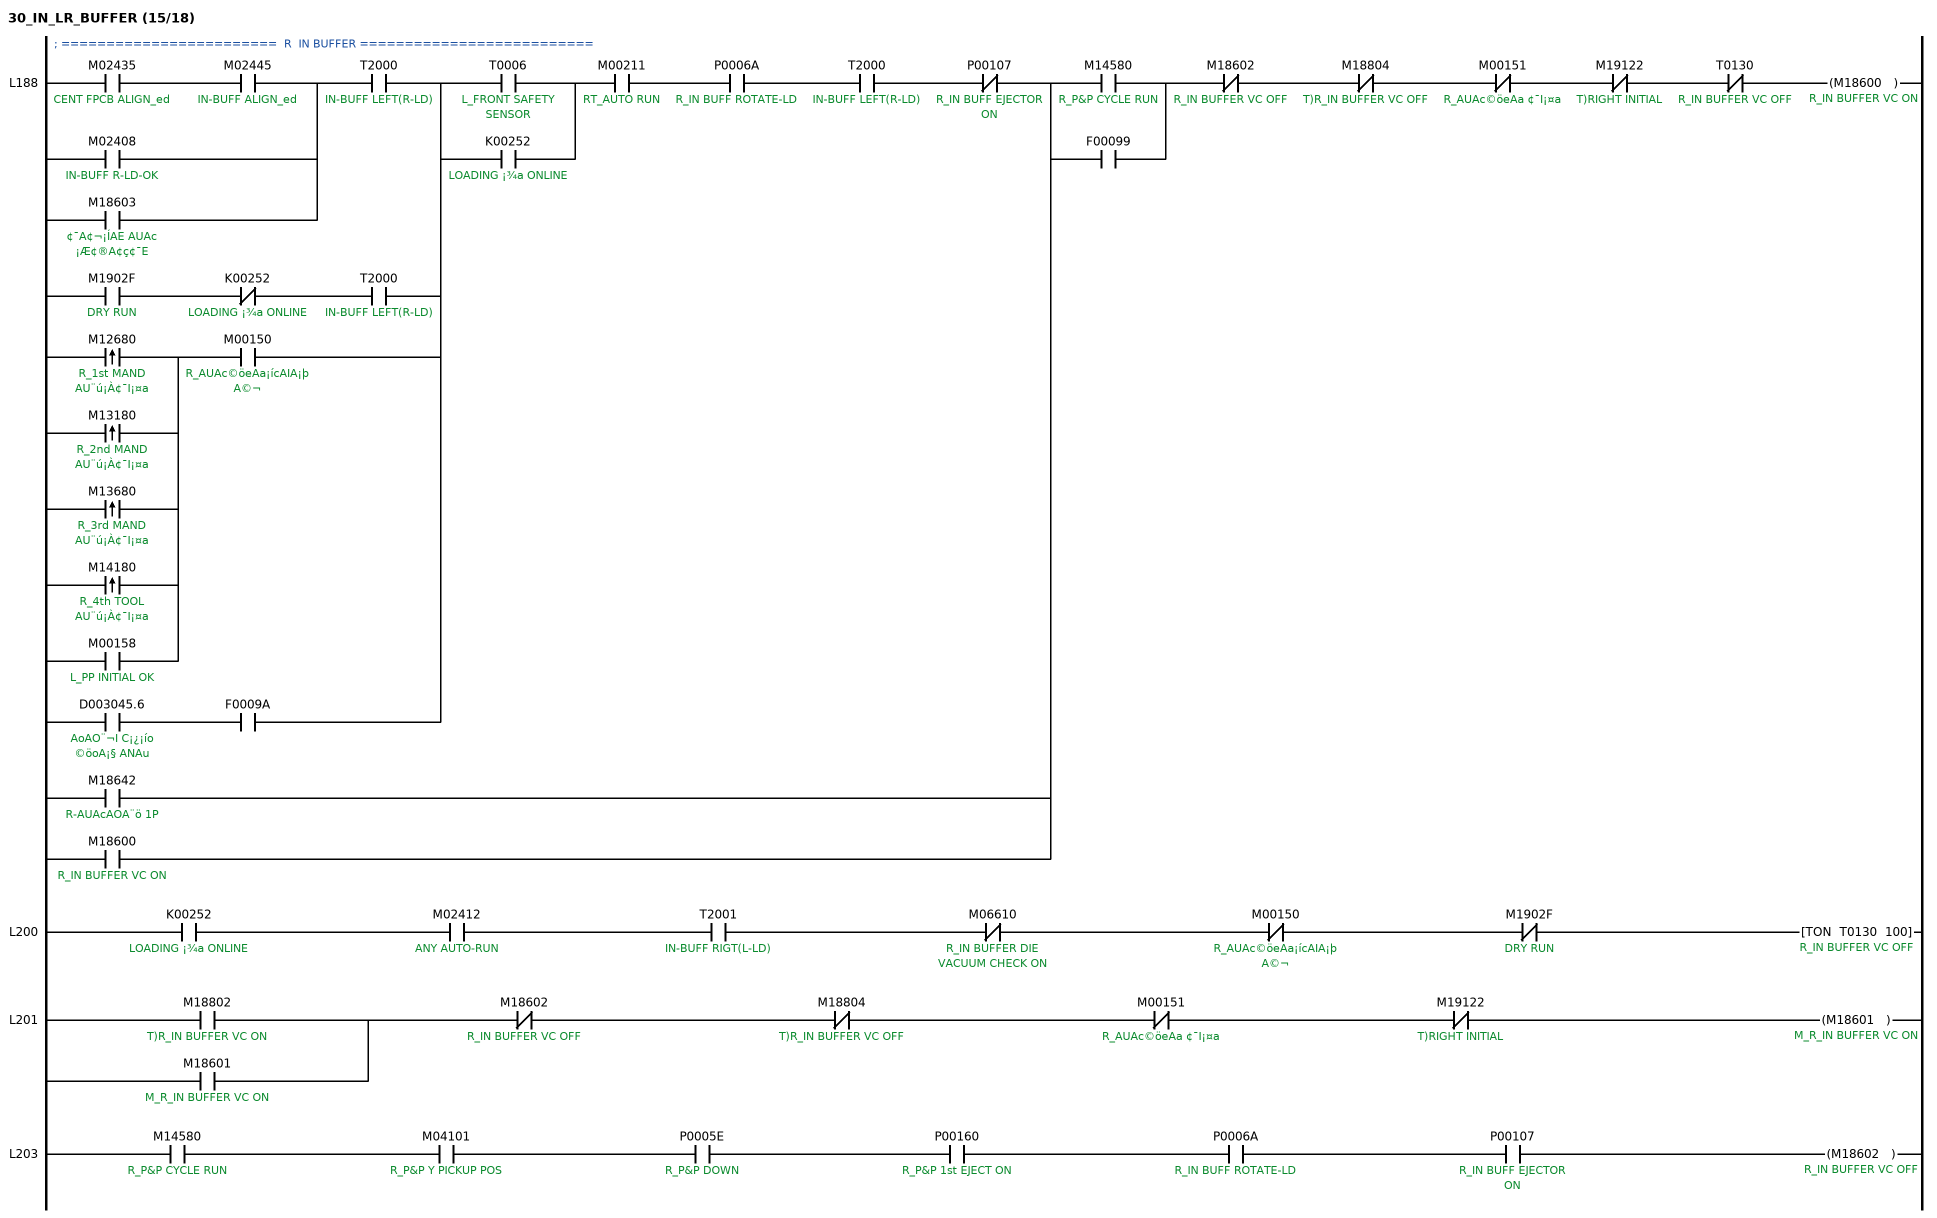
// ========================  R  IN BUFFER ==========================
; L188
LOAD      M02435	// CENT FPCB ALIGN_ed
AND       M02445	// IN-BUFF ALIGN_ed
OR        M02408	// IN-BUFF R-LD-OK
OR        M18603	// ¢¯A¢¬¡ÍAE AUAc ¡Æ¢®A¢ç¢¯E
AND       T2000	// IN-BUFF LEFT(R-LD)
LOAD      M1902F	// DRY RUN
AND NOT   K00252	// LOADING ¡¾a ONLINE
AND       T2000	// IN-BUFF LEFT(R-LD)
OR LOAD
LOADP     M12680	// R_1st MAND AU¨ú¡À¢¯I¡¤a
ORP       M13180	// R_2nd MAND AU¨ú¡À¢¯I¡¤a
ORP       M13680	// R_3rd MAND AU¨ú¡À¢¯I¡¤a
ORP       M14180	// R_4th TOOL AU¨ú¡À¢¯I¡¤a
OR        M00158	// L_PP INITIAL OK
AND       M00150	// R_AUAc©öeAa¡ícAIA¡þA©¬
OR LOAD
LOAD      D003045.6	// AoAO¨¬I C¡¿¡ío ©öoA¡§ ANAu
AND       F0009A
OR LOAD
LOAD      T0006	// L_FRONT SAFETY SENSOR
OR        K00252	// LOADING ¡¾a ONLINE
AND LOAD
AND       M00211	// RT_AUTO RUN
AND       P0006A	// R_IN BUFF ROTATE-LD
AND       T2000	// IN-BUFF LEFT(R-LD)
AND NOT   P00107	// R_IN BUFF EJECTOR ON
OR        M18642	// R-AUAcAOA¨ö 1P
OR        M18600	// R_IN BUFFER VC ON
LOAD      M14580	// R_P&P CYCLE RUN
OR        F00099
AND LOAD
AND NOT   M18602	// R_IN BUFFER VC OFF
AND NOT   M18804	// T)R_IN BUFFER VC OFF
AND NOT   M00151	// R_AUAc©öeAa ¢¯I¡¤a
AND NOT   M19122	// T)RIGHT INITIAL
AND NOT   T0130	// R_IN BUFFER VC OFF
OUT       M18600	// R_IN BUFFER VC ON
; L200
LOAD      K00252	// LOADING ¡¾a ONLINE
AND       M02412	// ANY AUTO-RUN
AND       T2001	// IN-BUFF RIGT(L-LD)
AND NOT   M06610	// R_IN BUFFER DIE VACUUM CHECK ON
AND NOT   M00150	// R_AUAc©öeAa¡ícAIA¡þA©¬
AND NOT   M1902F	// DRY RUN
TON       T0130 100	// R_IN BUFFER VC OFF
; L201
LOAD      M18802	// T)R_IN BUFFER VC ON
OR        M18601	// M_R_IN BUFFER VC ON
AND NOT   M18602	// R_IN BUFFER VC OFF
AND NOT   M18804	// T)R_IN BUFFER VC OFF
AND NOT   M00151	// R_AUAc©öeAa ¢¯I¡¤a
AND NOT   M19122	// T)RIGHT INITIAL
OUT       M18601	// M_R_IN BUFFER VC ON
; L203
LOAD      M14580	// R_P&P CYCLE RUN
AND       M04101	// R_P&P Y PICKUP POS
AND       P0005E	// R_P&P DOWN
AND       P00160	// R_P&P 1st EJECT ON
AND       P0006A	// R_IN BUFF ROTATE-LD
AND       P00107	// R_IN BUFF EJECTOR ON
OUT       M18602	// R_IN BUFFER VC OFF

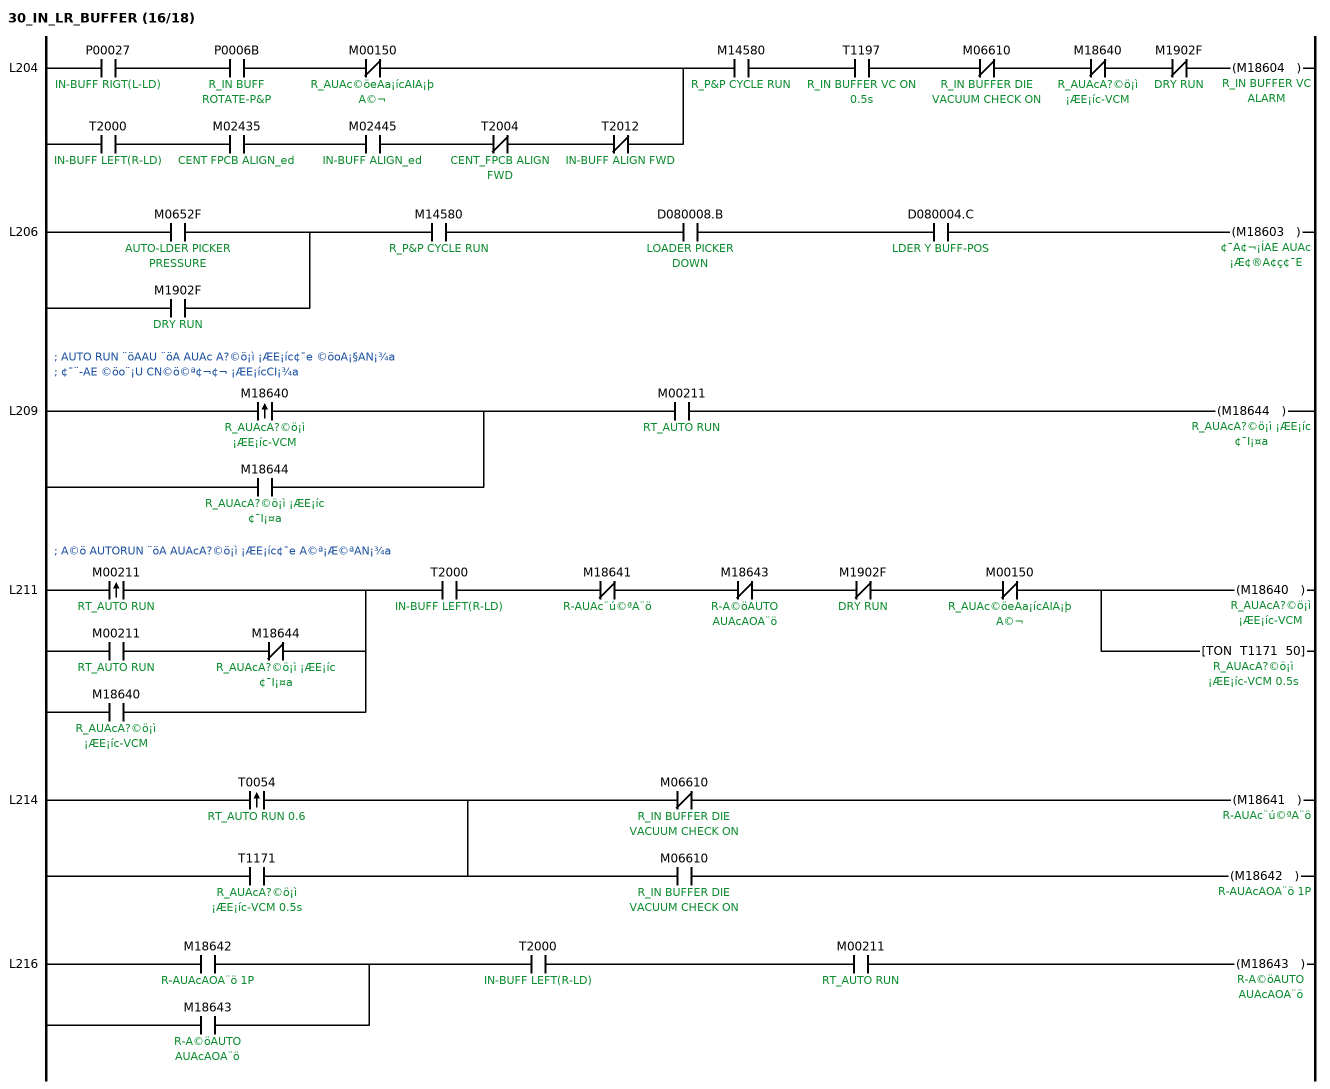
; L204
LOAD      P00027	// IN-BUFF RIGT(L-LD)
AND       P0006B	// R_IN BUFF ROTATE-P&P
AND NOT   M00150	// R_AUAc©öeAa¡ícAIA¡þA©¬
LOAD      T2000	// IN-BUFF LEFT(R-LD)
AND       M02435	// CENT FPCB ALIGN_ed
AND       M02445	// IN-BUFF ALIGN_ed
AND NOT   T2004	// CENT_FPCB ALIGN FWD
AND NOT   T2012	// IN-BUFF ALIGN FWD
OR LOAD
AND       M14580	// R_P&P CYCLE RUN
AND       T1197	// R_IN BUFFER VC ON 0.5s
AND NOT   M06610	// R_IN BUFFER DIE VACUUM CHECK ON
AND NOT   M18640	// R_AUAcA?©ö¡ì ¡ÆE¡íc-VCM
AND NOT   M1902F	// DRY RUN
OUT       M18604	// R_IN BUFFER VC ALARM
; L206
LOAD      M0652F	// AUTO-LDER PICKER PRESSURE
OR        M1902F	// DRY RUN
AND       M14580	// R_P&P CYCLE RUN
AND       D080008.B	// LOADER PICKER DOWN
AND       D080004.C	// LDER Y BUFF-POS
OUT       M18603	// ¢¯A¢¬¡ÍAE AUAc ¡Æ¢®A¢ç¢¯E
// AUTO RUN ¨öAAU ¨öA AUAc A?©ö¡ì ¡ÆE¡íc¢¯e ©öoA¡§AN¡¾a
; L209
LOADP     M18640	// R_AUAcA?©ö¡ì ¡ÆE¡íc-VCM
OR        M18644	// R_AUAcA?©ö¡ì ¡ÆE¡íc ¢¯I¡¤a
AND       M00211	// RT_AUTO RUN
OUT       M18644	// R_AUAcA?©ö¡ì ¡ÆE¡íc ¢¯I¡¤a
// output comment: ¢¯¨­AE ©öo¨¡U CN©ö©ª¢¬¢¬ ¡ÆE¡ícCI¡¾a
; L211
LOADP     M00211	// RT_AUTO RUN
LOAD      M00211	// RT_AUTO RUN
AND NOT   M18644	// R_AUAcA?©ö¡ì ¡ÆE¡íc ¢¯I¡¤a
OR LOAD
OR        M18640	// R_AUAcA?©ö¡ì ¡ÆE¡íc-VCM
AND       T2000	// IN-BUFF LEFT(R-LD)
AND NOT   M18641	// R-AUAc¨ú©ªA¨ö
AND NOT   M18643	// R-A©öAUTO AUAcAOA¨ö
AND NOT   M1902F	// DRY RUN
AND NOT   M00150	// R_AUAc©öeAa¡ícAIA¡þA©¬
OUT       M18640	// R_AUAcA?©ö¡ì ¡ÆE¡íc-VCM
TON       T1171 50	// R_AUAcA?©ö¡ì ¡ÆE¡íc-VCM 0.5s
// output comment: A©ö AUTORUN ¨öA AUAcA?©ö¡ì ¡ÆE¡íc¢¯e A©ª¡Æ©ªAN¡¾a
; L214
LOADP     T0054	// RT_AUTO RUN 0.6
OR        T1171	// R_AUAcA?©ö¡ì ¡ÆE¡íc-VCM 0.5s
MPUSH
AND NOT   M06610	// R_IN BUFFER DIE VACUUM CHECK ON
OUT       M18641	// R-AUAc¨ú©ªA¨ö
MPOP
AND       M06610	// R_IN BUFFER DIE VACUUM CHECK ON
OUT       M18642	// R-AUAcAOA¨ö 1P
; L216
LOAD      M18642	// R-AUAcAOA¨ö 1P
OR        M18643	// R-A©öAUTO AUAcAOA¨ö
AND       T2000	// IN-BUFF LEFT(R-LD)
AND       M00211	// RT_AUTO RUN
OUT       M18643	// R-A©öAUTO AUAcAOA¨ö

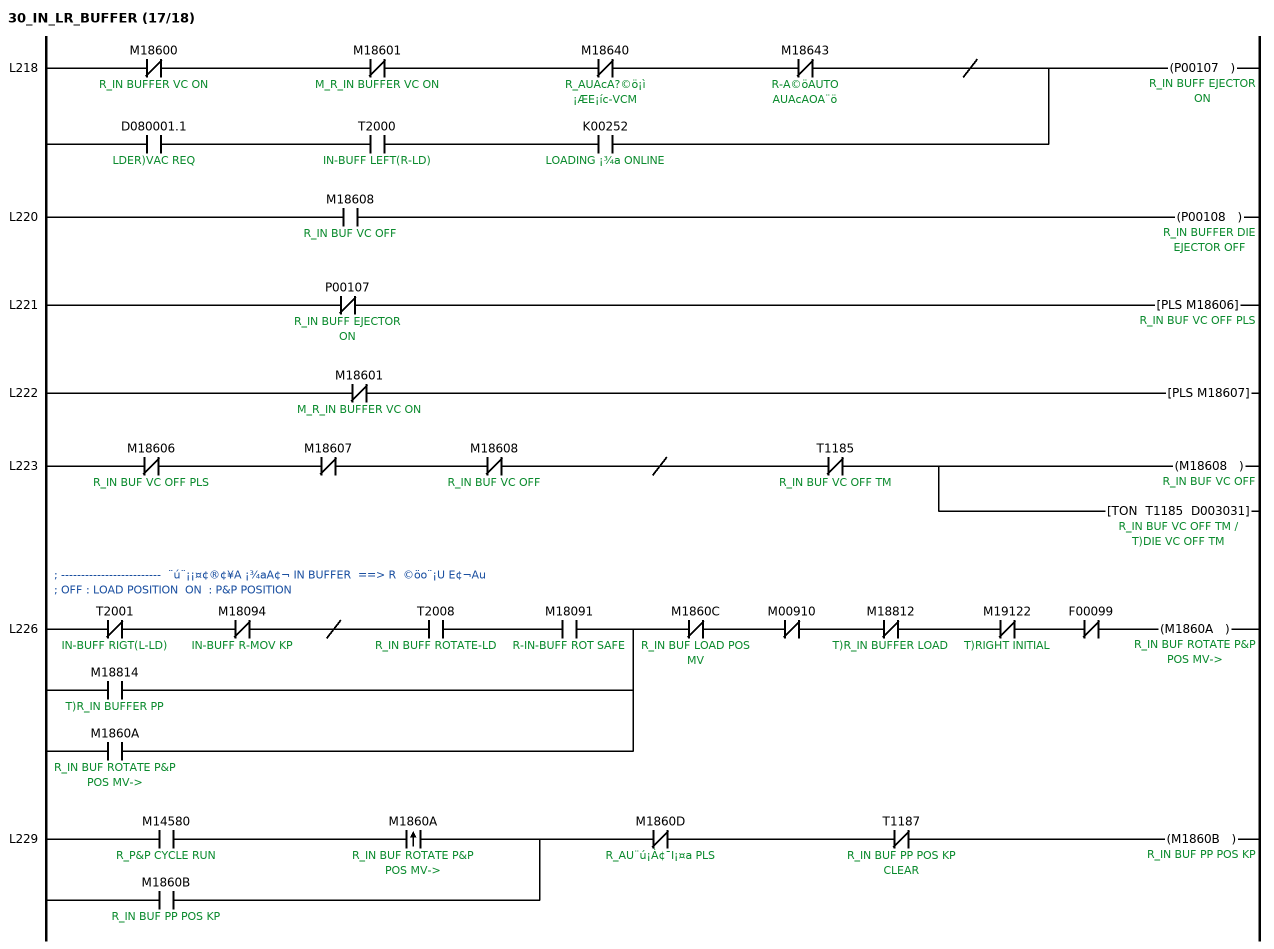
; L218
LOAD NOT  M18600	// R_IN BUFFER VC ON
AND NOT   M18601	// M_R_IN BUFFER VC ON
AND NOT   M18640	// R_AUAcA?©ö¡ì ¡ÆE¡íc-VCM
AND NOT   M18643	// R-A©öAUTO AUAcAOA¨ö
NOT
LOAD      D080001.1	// LDER)VAC REQ
AND       T2000	// IN-BUFF LEFT(R-LD)
AND       K00252	// LOADING ¡¾a ONLINE
OR LOAD
OUT       P00107	// R_IN BUFF EJECTOR ON
; L220
LOAD      M18608	// R_IN BUF VC OFF
OUT       P00108	// R_IN BUFFER DIE EJECTOR OFF
; L221
LOAD NOT  P00107	// R_IN BUFF EJECTOR ON
OUTP      M18606	// R_IN BUF VC OFF PLS
; L222
LOAD NOT  M18601	// M_R_IN BUFFER VC ON
OUTP      M18607
; L223
LOAD NOT  M18606	// R_IN BUF VC OFF PLS
AND NOT   M18607
AND NOT   M18608	// R_IN BUF VC OFF
NOT
AND NOT   T1185	// R_IN BUF VC OFF TM
OUT       M18608	// R_IN BUF VC OFF
TON       T1185 D003031	// R_IN BUF VC OFF TM / T)DIE VC OFF TM
// -------------------------  ¨ú¨¡¡¤¢®¢¥A ¡¾aA¢¬ IN BUFFER  ==> R  ©öo¨¡U E¢¬Au
; L226
LOAD NOT  T2001	// IN-BUFF RIGT(L-LD)
AND NOT   M18094	// IN-BUFF R-MOV KP
NOT
AND       T2008	// R_IN BUFF ROTATE-LD
AND       M18091	// R-IN-BUFF ROT SAFE
OR        M18814	// T)R_IN BUFFER PP
OR        M1860A	// R_IN BUF ROTATE P&P POS MV->
AND NOT   M1860C	// R_IN BUF LOAD POS MV
AND NOT   M00910
AND NOT   M18812	// T)R_IN BUFFER LOAD
AND NOT   M19122	// T)RIGHT INITIAL
AND NOT   F00099
OUT       M1860A	// R_IN BUF ROTATE P&P POS MV->
// output comment: OFF : LOAD POSITION  ON  : P&P POSITION
; L229
LOAD      M14580	// R_P&P CYCLE RUN
ANDP      M1860A	// R_IN BUF ROTATE P&P POS MV->
OR        M1860B	// R_IN BUF PP POS KP
AND NOT   M1860D	// R_AU¨ú¡À¢¯I¡¤a PLS
AND NOT   T1187	// R_IN BUF PP POS KP CLEAR
OUT       M1860B	// R_IN BUF PP POS KP

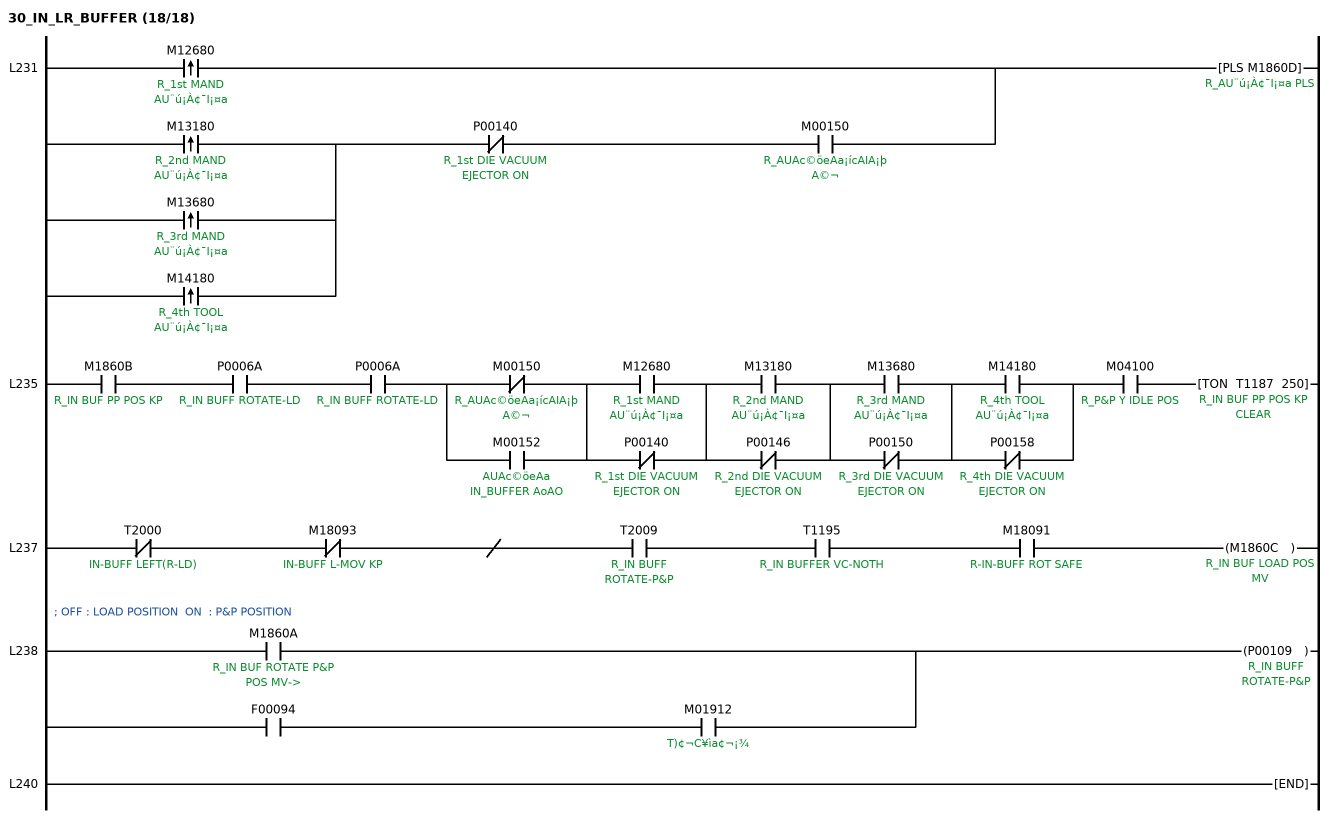
; L231
LOADP     M12680	// R_1st MAND AU¨ú¡À¢¯I¡¤a
LOADP     M13180	// R_2nd MAND AU¨ú¡À¢¯I¡¤a
ORP       M13680	// R_3rd MAND AU¨ú¡À¢¯I¡¤a
ORP       M14180	// R_4th TOOL AU¨ú¡À¢¯I¡¤a
AND NOT   P00140	// R_1st DIE VACUUM EJECTOR ON
AND       M00150	// R_AUAc©öeAa¡ícAIA¡þA©¬
OR LOAD
OUTP      M1860D	// R_AU¨ú¡À¢¯I¡¤a PLS
; L235
LOAD      M1860B	// R_IN BUF PP POS KP
AND       P0006A	// R_IN BUFF ROTATE-LD
AND       P0006A	// R_IN BUFF ROTATE-LD
LOAD NOT  M00150	// R_AUAc©öeAa¡ícAIA¡þA©¬
OR        M00152	// AUAc©öeAa IN_BUFFER AoAO 
AND LOAD
LOAD      M12680	// R_1st MAND AU¨ú¡À¢¯I¡¤a
OR NOT    P00140	// R_1st DIE VACUUM EJECTOR ON
AND LOAD
LOAD      M13180	// R_2nd MAND AU¨ú¡À¢¯I¡¤a
OR NOT    P00146	// R_2nd DIE VACUUM EJECTOR ON
AND LOAD
LOAD      M13680	// R_3rd MAND AU¨ú¡À¢¯I¡¤a
OR NOT    P00150	// R_3rd DIE VACUUM EJECTOR ON
AND LOAD
LOAD      M14180	// R_4th TOOL AU¨ú¡À¢¯I¡¤a
OR NOT    P00158	// R_4th DIE VACUUM EJECTOR ON
AND LOAD
AND       M04100	// R_P&P Y IDLE POS
TON       T1187 250	// R_IN BUF PP POS KP CLEAR
; L237
LOAD NOT  T2000	// IN-BUFF LEFT(R-LD)
AND NOT   M18093	// IN-BUFF L-MOV KP
NOT
AND       T2009	// R_IN BUFF ROTATE-P&P
AND       T1195	// R_IN BUFFER VC-NOTH
AND       M18091	// R-IN-BUFF ROT SAFE
OUT       M1860C	// R_IN BUF LOAD POS MV
; L238
LOAD      M1860A	// R_IN BUF ROTATE P&P POS MV->
LOAD      F00094
AND       M01912	// T)¢¬C¥ìa¢¬¡¾
OR LOAD
OUT       P00109	// R_IN BUFF ROTATE-P&P
// output comment: OFF : LOAD POSITION  ON  : P&P POSITION
; L240
END

PROGRAM 31_OUT_LR_BUFFER (task: ¨ö¨¬A¥ì CA¡¤I¡¾¡¿¡¤¡Í)

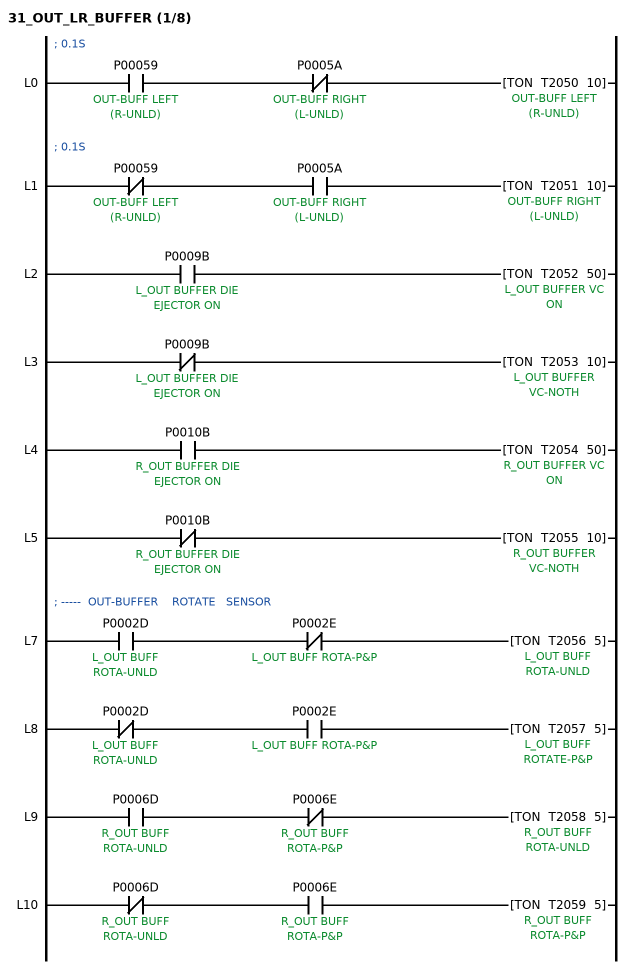
; L0
LOAD      P00059	// OUT-BUFF LEFT (R-UNLD)
AND NOT   P0005A	// OUT-BUFF RIGHT (L-UNLD)
TON       T2050 10	// OUT-BUFF LEFT (R-UNLD)
// output comment: 0.1S
; L1
LOAD NOT  P00059	// OUT-BUFF LEFT (R-UNLD)
AND       P0005A	// OUT-BUFF RIGHT (L-UNLD)
TON       T2051 10	// OUT-BUFF RIGHT (L-UNLD)
// output comment: 0.1S
; L2
LOAD      P0009B	// L_OUT BUFFER DIE EJECTOR ON
TON       T2052 50	// L_OUT BUFFER VC ON
; L3
LOAD NOT  P0009B	// L_OUT BUFFER DIE EJECTOR ON
TON       T2053 10	// L_OUT BUFFER VC-NOTH
; L4
LOAD      P0010B	// R_OUT BUFFER DIE EJECTOR ON
TON       T2054 50	// R_OUT BUFFER VC ON
; L5
LOAD NOT  P0010B	// R_OUT BUFFER DIE EJECTOR ON
TON       T2055 10	// R_OUT BUFFER VC-NOTH
// -----  OUT-BUFFER    ROTATE   SENSOR
; L7
LOAD      P0002D	// L_OUT BUFF ROTA-UNLD
AND NOT   P0002E	// L_OUT BUFF ROTA-P&P
TON       T2056 5	// L_OUT BUFF ROTA-UNLD
; L8
LOAD NOT  P0002D	// L_OUT BUFF ROTA-UNLD
AND       P0002E	// L_OUT BUFF ROTA-P&P
TON       T2057 5	// L_OUT BUFF ROTATE-P&P
; L9
LOAD      P0006D	// R_OUT BUFF ROTA-UNLD
AND NOT   P0006E	// R_OUT BUFF ROTA-P&P
TON       T2058 5	// R_OUT BUFF ROTA-UNLD
; L10
LOAD NOT  P0006D	// R_OUT BUFF ROTA-UNLD
AND       P0006E	// R_OUT BUFF ROTA-P&P
TON       T2059 5	// R_OUT BUFF ROTA-P&P

